ABB RAPID module: PPFP_hurdleJumps

MODULE Weld_ALL_OF_THE_Channels_PR3


    ! NOTES
    ! 6/18/18  CHANGED THE LRnRL_CHAN SETTER's FORLOOP TO START @ 1, WAS MISSING ON M-55's
    ! 3/25/19 CHANGED LL/RR GENERIC STITCH TO SKIP WELD 1 IF ITS A TIGHT BOX
    !  ALSO MADE CHANGES TO THE LRnRL_CHANPLAN, THE_OBJECT = "Push_Stop",   3RD IF TO MAKE THE WELD FLIP IF THE WELD START WAS IN THE MIDDLE OF THE PUSHSTOP
    ! R23  ADDED SR_X2_Y3.TRANS.Y TO THE HURDLES.  TO ALLOW SOME WIGGLE ROOM WHILE TACKING UP, AND STILL BE ABLE TO HOP THE FENCES.
    ! R27 Changed " LRnRL_CHAN_PLAN "Y4"; " FROM "IF (THE_OBJECT = "Y3" AND HORIZ_Y3 <> FP_Height) OR ( THE_OBJECT = "Y4" AND HORIZ_Y4 <> FP_Height) THEN"  TO "IF (THE_OBJECT = "Y3" AND HORIZ_Y3 <> FP_Height) OR ( THE_OBJECT = "Y4" AND HORIZ_Y4 = FP_Height) THEN"
	! 10/21/19 SS
    !  ADDED  " and MY3_Weld_Count > 0 THEN " TO KEEP THE WELD FROM BEING FLIPPED OVER WHEN THERE IS NO CENTER BAR 6/3/20 SS

	! CHANGED PLAN_dUH_cHAN, WHEN W=7, FOR PUSH_STOP = 303,ON 6894640 WAS CRASHING 10/20/20/SS

	! Changed the arrays from 35 to 40, ran out of welds, gave error.  7/22/21/SS

    ! UpDated 7/22/21/SS skipping all weld below the anchor on LRnRL, just to satisify the need of having a AngleIron inside the FP 6898779 on a Friday when I'm not here and Dan W. will just walk away.

PERS robtarget RL_Chan_goingUP:=[[248.58,439.22,15.69],[0.0743186,0.868569,0.302507,0.385428],[0,1,-2,0],[9E+09,-45,0.00451687,9E+09,9E+09,9E+09]];
PERS robtarget RL_Chan_goingUPcorner:=[[248.57,468.99,15.69],[0.00441198,0.818231,0.408605,0.404377],[0,1,-2,0],[9E+09,-40,-5,9E+09,9E+09,9E+09]];

PERS robtarget RL_Chan_goingDOWN:=[[248.55,439.20,15.69],[0.166009,0.884241,0.263964,0.347682],[0,1,-2,0],[9E+09,-45,0.00435694,9E+09,9E+09,9E+09]];
PERS robtarget RL_Chan_BOTTOMcorner:=[[248.55,408.61,15.69],[0.263807,0.884566,0.230134,0.308201],[0,1,-2,0],[9E+09,-40,5.00001,9E+09,9E+09,9E+09]];

PERS robtarget RL_CHANFLAT_goingup:=[[223.12,483.90,15.69],[0.0686406,0.860922,0.436323,0.252434],[0,1,-2,0],[9E+09,-30,0.00345066,9E+09,9E+09,9E+09]];
PERS robtarget RL_CHANFLAT_TOPcorner:=[[223.12,483.90,15.69],[0.0592125,-0.838583,-0.451769,-0.298627],[0,1,-2,0],[9E+09,-25,-4.99996,9E+09,9E+09,9E+09]];

PERS robtarget LL_CHAN_GoingUp:=[[-270.37,436.99,15.21],[0.144124,0.788012,0.487648,0.347081],[0,0,-2,0],[9E+09,-45,0.00410816,9E+09,9E+09,9E+09]];
PERS robtarget LL_CHAN_goingupcorner:=[[-265.50,887.94,15.22],[0.0140209,0.753344,0.518535,0.404224],[-1,0,-1,0],[9E+09,-40,-5,9E+09,9E+09,9E+09]];

PERS robtarget LL_CHAN_GOINGdown:=[[-270.37,436.99,15.21],[0.22246,0.805806,0.454482,0.307627],[0,0,-2,0],[9E+09,-45,0.00410816,9E+09,9E+09,9E+09]];
PERS robtarget LL_CHAN_GOINGdowncorner:=[[-270.36,411.33,15.20],[0.297563,0.81565,0.425985,0.254378],[0,0,-2,0],[9E+09,-40,4.99995,9E+09,9E+09,9E+09]];


PERS robtarget RR_CHAN_GOINGup:=[[265.74,425.05,15.18],[0.346334,0.329821,-0.862433,-0.165773],[-1,0,-2,0],[9E+09,-45,180,9E+09,9E+09,9E+09]];
PERS robtarget RR_CHAN_TOPcorner:=[[265.70,886.67,15.16],[0.257593,0.29389,-0.878079,-0.276138],[-1,0,-2,0],[9E+09,-40,185,9E+09,9E+09,9E+09]];

PERS robtarget RR_CHAN_GOINGdown:=[[269.75,437.02,16.58],[0.403142,0.332329,-0.846748,-0.100255],[-1,0,-2,0],[9E+09,-45,180,9E+09,9E+09,9E+09]];
PERS robtarget RR_CHAN_BOTTOMcorner:=[[269.76,437.02,16.58],[0.430288,0.36564,-0.825086,0.0198048],[-1,0,-1,0],[9E+09,-40,175,9E+09,9E+09,9E+09]];

PERS robtarget LR_CHAN_GOINGup:=[[-249.44,441.38,17.56],[0.34969,0.292965,-0.875927,-0.156972],[-1,0,-2,0],[9E+09,-45,180,9E+09,9E+09,9E+09]];
PERS robtarget LR_CHAN_goingup_corner:=[[-249.44,441.36,17.56],[0.332557,0.268512,-0.875476,-0.225495],[-1,0,-2,0],[9E+09,-40,185,9E+09,9E+09,9E+09]];

PERS robtarget LR_CHAN_GOINGdown:=[[-249.43,441.36,17.56],[0.393213,0.316458,-0.858163,-0.0937788],[-1,0,-2,0],[9E+09,-45,180,9E+09,9E+09,9E+09]];
PERS robtarget LR_CHAN_goingdown_corner:=[[-249.43,441.35,17.56],[0.431123,0.340521,-0.835569,0.0017755],[-1,0,-2,0],[9E+09,-40,175,9E+09,9E+09,9E+09]];

PERS robtarget LR_CHANFLAT_GOINGup:=[[-225.09,482.69,17.56],[0.267219,0.316082,-0.899666,-0.138875],[-1,0,-2,0],[9E+09,-30,180,9E+09,9E+09,9E+09]];
PERS robtarget LR_CHANFLAT_GOINGupcorner:=[[-225.09,482.69,17.56],[0.224093,0.303126,-0.899516,-0.220836],[-1,0,-2,0],[9E+09,-25,185,9E+09,9E+09,9E+09]];




VAR robtarget LL_CHAN_WELDS{40,3}:=[[ [[184.43,695.20,80.98],[0.0842675,0.873996,0.3985,0.265006],[0,0,0,0],[9E+09,-30,0.00423255,9E+09,9E+09,9E+09]],[[184.43,695.20,80.98],[0.0842675,0.873996,0.3985,0.265006],[0,0,0,0],[9E+09,-30,0.00423255,9E+09,9E+09,9E+09]],[[184.43,695.20,80.98],[0.0842675,0.873996,0.3985,0.265006],[0,0,0,0],[9E+09,-30,0.00423255,9E+09,9E+09,9E+09]]],
     [[[184.43,695.20,80.98],[0.0842675,0.873996,0.3985,0.265006],[0,0,0,0],[9E+09,-30,0.00423255,9E+09,9E+09,9E+09]],[[184.43,695.20,80.98],[0.0842675,0.873996,0.3985,0.265006],[0,0,0,0],[9E+09,-30,0.00423255,9E+09,9E+09,9E+09]],[[184.43,695.20,80.98],[0.0842675,0.873996,0.3985,0.265006],[0,0,0,0],[9E+09,-30,0.00423255,9E+09,9E+09,9E+09]]],
     [[[184.43,695.20,80.98],[0.0842675,0.873996,0.3985,0.265006],[0,0,0,0],[9E+09,-30,0.00423255,9E+09,9E+09,9E+09]],[[184.43,695.20,80.98],[0.0842675,0.873996,0.3985,0.265006],[0,0,0,0],[9E+09,-30,0.00423255,9E+09,9E+09,9E+09]],[[184.43,695.20,80.98],[0.0842675,0.873996,0.3985,0.265006],[0,0,0,0],[9E+09,-30,0.00423255,9E+09,9E+09,9E+09]]],
     [[[184.43,695.20,80.98],[0.0842675,0.873996,0.3985,0.265006],[0,0,0,0],[9E+09,-30,0.00423255,9E+09,9E+09,9E+09]],[[184.43,695.20,80.98],[0.0842675,0.873996,0.3985,0.265006],[0,0,0,0],[9E+09,-30,0.00423255,9E+09,9E+09,9E+09]],[[184.43,695.20,80.98],[0.0842675,0.873996,0.3985,0.265006],[0,0,0,0],[9E+09,-30,0.00423255,9E+09,9E+09,9E+09]]],
     [[[184.43,695.20,80.98],[0.0842675,0.873996,0.3985,0.265006],[0,0,0,0],[9E+09,-30,0.00423255,9E+09,9E+09,9E+09]],[[184.43,695.20,80.98],[0.0842675,0.873996,0.3985,0.265006],[0,0,0,0],[9E+09,-30,0.00423255,9E+09,9E+09,9E+09]],[[184.43,695.20,80.98],[0.0842675,0.873996,0.3985,0.265006],[0,0,0,0],[9E+09,-30,0.00423255,9E+09,9E+09,9E+09]]],
     [[[184.43,695.20,80.98],[0.0842675,0.873996,0.3985,0.265006],[0,0,0,0],[9E+09,-30,0.00423255,9E+09,9E+09,9E+09]],[[184.43,695.20,80.98],[0.0842675,0.873996,0.3985,0.265006],[0,0,0,0],[9E+09,-30,0.00423255,9E+09,9E+09,9E+09]],[[184.43,695.20,80.98],[0.0842675,0.873996,0.3985,0.265006],[0,0,0,0],[9E+09,-30,0.00423255,9E+09,9E+09,9E+09]]],
     [[[184.43,695.20,80.98],[0.0842675,0.873996,0.3985,0.265006],[0,0,0,0],[9E+09,-30,0.00423255,9E+09,9E+09,9E+09]],[[184.43,695.20,80.98],[0.0842675,0.873996,0.3985,0.265006],[0,0,0,0],[9E+09,-30,0.00423255,9E+09,9E+09,9E+09]],[[184.43,695.20,80.98],[0.0842675,0.873996,0.3985,0.265006],[0,0,0,0],[9E+09,-30,0.00423255,9E+09,9E+09,9E+09]]],
     [[[184.43,695.20,80.98],[0.0842675,0.873996,0.3985,0.265006],[0,0,0,0],[9E+09,-30,0.00423255,9E+09,9E+09,9E+09]],[[184.43,695.20,80.98],[0.0842675,0.873996,0.3985,0.265006],[0,0,0,0],[9E+09,-30,0.00423255,9E+09,9E+09,9E+09]],[[184.43,695.20,80.98],[0.0842675,0.873996,0.3985,0.265006],[0,0,0,0],[9E+09,-30,0.00423255,9E+09,9E+09,9E+09]]],
     [[[184.43,695.20,80.98],[0.0842675,0.873996,0.3985,0.265006],[0,0,0,0],[9E+09,-30,0.00423255,9E+09,9E+09,9E+09]],[[184.43,695.20,80.98],[0.0842675,0.873996,0.3985,0.265006],[0,0,0,0],[9E+09,-30,0.00423255,9E+09,9E+09,9E+09]],[[184.43,695.20,80.98],[0.0842675,0.873996,0.3985,0.265006],[0,0,0,0],[9E+09,-30,0.00423255,9E+09,9E+09,9E+09]]],
     [[[184.43,695.20,80.98],[0.0842675,0.873996,0.3985,0.265006],[0,0,0,0],[9E+09,-30,0.00423255,9E+09,9E+09,9E+09]],[[184.43,695.20,80.98],[0.0842675,0.873996,0.3985,0.265006],[0,0,0,0],[9E+09,-30,0.00423255,9E+09,9E+09,9E+09]],[[184.43,695.20,80.98],[0.0842675,0.873996,0.3985,0.265006],[0,0,0,0],[9E+09,-30,0.00423255,9E+09,9E+09,9E+09]]],
     [[[184.43,695.20,80.98],[0.0842675,0.873996,0.3985,0.265006],[0,0,0,0],[9E+09,-30,0.00423255,9E+09,9E+09,9E+09]],[[184.43,695.20,80.98],[0.0842675,0.873996,0.3985,0.265006],[0,0,0,0],[9E+09,-30,0.00423255,9E+09,9E+09,9E+09]],[[184.43,695.20,80.98],[0.0842675,0.873996,0.3985,0.265006],[0,0,0,0],[9E+09,-30,0.00423255,9E+09,9E+09,9E+09]]],
     [[[184.43,695.20,80.98],[0.0842675,0.873996,0.3985,0.265006],[0,0,0,0],[9E+09,-30,0.00423255,9E+09,9E+09,9E+09]],[[184.43,695.20,80.98],[0.0842675,0.873996,0.3985,0.265006],[0,0,0,0],[9E+09,-30,0.00423255,9E+09,9E+09,9E+09]],[[184.43,695.20,80.98],[0.0842675,0.873996,0.3985,0.265006],[0,0,0,0],[9E+09,-30,0.00423255,9E+09,9E+09,9E+09]]],
     [[[184.43,695.20,80.98],[0.0842675,0.873996,0.3985,0.265006],[0,0,0,0],[9E+09,-30,0.00423255,9E+09,9E+09,9E+09]],[[184.43,695.20,80.98],[0.0842675,0.873996,0.3985,0.265006],[0,0,0,0],[9E+09,-30,0.00423255,9E+09,9E+09,9E+09]],[[184.43,695.20,80.98],[0.0842675,0.873996,0.3985,0.265006],[0,0,0,0],[9E+09,-30,0.00423255,9E+09,9E+09,9E+09]]],
     [[[184.43,695.20,80.98],[0.0842675,0.873996,0.3985,0.265006],[0,0,0,0],[9E+09,-30,0.00423255,9E+09,9E+09,9E+09]],[[184.43,695.20,80.98],[0.0842675,0.873996,0.3985,0.265006],[0,0,0,0],[9E+09,-30,0.00423255,9E+09,9E+09,9E+09]],[[184.43,695.20,80.98],[0.0842675,0.873996,0.3985,0.265006],[0,0,0,0],[9E+09,-30,0.00423255,9E+09,9E+09,9E+09]]],
     [[[184.43,695.20,80.98],[0.0842675,0.873996,0.3985,0.265006],[0,0,0,0],[9E+09,-30,0.00423255,9E+09,9E+09,9E+09]],[[184.43,695.20,80.98],[0.0842675,0.873996,0.3985,0.265006],[0,0,0,0],[9E+09,-30,0.00423255,9E+09,9E+09,9E+09]],[[184.43,695.20,80.98],[0.0842675,0.873996,0.3985,0.265006],[0,0,0,0],[9E+09,-30,0.00423255,9E+09,9E+09,9E+09]]],
     [[[184.43,695.20,80.98],[0.0842675,0.873996,0.3985,0.265006],[0,0,0,0],[9E+09,-30,0.00423255,9E+09,9E+09,9E+09]],[[184.43,695.20,80.98],[0.0842675,0.873996,0.3985,0.265006],[0,0,0,0],[9E+09,-30,0.00423255,9E+09,9E+09,9E+09]],[[184.43,695.20,80.98],[0.0842675,0.873996,0.3985,0.265006],[0,0,0,0],[9E+09,-30,0.00423255,9E+09,9E+09,9E+09]]],
     [[[184.43,695.20,80.98],[0.0842675,0.873996,0.3985,0.265006],[0,0,0,0],[9E+09,-30,0.00423255,9E+09,9E+09,9E+09]],[[184.43,695.20,80.98],[0.0842675,0.873996,0.3985,0.265006],[0,0,0,0],[9E+09,-30,0.00423255,9E+09,9E+09,9E+09]],[[184.43,695.20,80.98],[0.0842675,0.873996,0.3985,0.265006],[0,0,0,0],[9E+09,-30,0.00423255,9E+09,9E+09,9E+09]]],
     [[[184.43,695.20,80.98],[0.0842675,0.873996,0.3985,0.265006],[0,0,0,0],[9E+09,-30,0.00423255,9E+09,9E+09,9E+09]],[[184.43,695.20,80.98],[0.0842675,0.873996,0.3985,0.265006],[0,0,0,0],[9E+09,-30,0.00423255,9E+09,9E+09,9E+09]],[[184.43,695.20,80.98],[0.0842675,0.873996,0.3985,0.265006],[0,0,0,0],[9E+09,-30,0.00423255,9E+09,9E+09,9E+09]]],
     [[[184.43,695.20,80.98],[0.0842675,0.873996,0.3985,0.265006],[0,0,0,0],[9E+09,-30,0.00423255,9E+09,9E+09,9E+09]],[[184.43,695.20,80.98],[0.0842675,0.873996,0.3985,0.265006],[0,0,0,0],[9E+09,-30,0.00423255,9E+09,9E+09,9E+09]],[[184.43,695.20,80.98],[0.0842675,0.873996,0.3985,0.265006],[0,0,0,0],[9E+09,-30,0.00423255,9E+09,9E+09,9E+09]]],
     [[[184.43,695.20,80.98],[0.0842675,0.873996,0.3985,0.265006],[0,0,0,0],[9E+09,-30,0.00423255,9E+09,9E+09,9E+09]],[[184.43,695.20,80.98],[0.0842675,0.873996,0.3985,0.265006],[0,0,0,0],[9E+09,-30,0.00423255,9E+09,9E+09,9E+09]],[[184.43,695.20,80.98],[0.0842675,0.873996,0.3985,0.265006],[0,0,0,0],[9E+09,-30,0.00423255,9E+09,9E+09,9E+09]]],
     [[[184.43,695.20,80.98],[0.0842675,0.873996,0.3985,0.265006],[0,0,0,0],[9E+09,-30,0.00423255,9E+09,9E+09,9E+09]],[[184.43,695.20,80.98],[0.0842675,0.873996,0.3985,0.265006],[0,0,0,0],[9E+09,-30,0.00423255,9E+09,9E+09,9E+09]],[[184.43,695.20,80.98],[0.0842675,0.873996,0.3985,0.265006],[0,0,0,0],[9E+09,-30,0.00423255,9E+09,9E+09,9E+09]]],
     [[[184.43,695.20,80.98],[0.0842675,0.873996,0.3985,0.265006],[0,0,0,0],[9E+09,-30,0.00423255,9E+09,9E+09,9E+09]],[[184.43,695.20,80.98],[0.0842675,0.873996,0.3985,0.265006],[0,0,0,0],[9E+09,-30,0.00423255,9E+09,9E+09,9E+09]],[[184.43,695.20,80.98],[0.0842675,0.873996,0.3985,0.265006],[0,0,0,0],[9E+09,-30,0.00423255,9E+09,9E+09,9E+09]]],
     [[[184.43,695.20,80.98],[0.0842675,0.873996,0.3985,0.265006],[0,0,0,0],[9E+09,-30,0.00423255,9E+09,9E+09,9E+09]],[[184.43,695.20,80.98],[0.0842675,0.873996,0.3985,0.265006],[0,0,0,0],[9E+09,-30,0.00423255,9E+09,9E+09,9E+09]],[[184.43,695.20,80.98],[0.0842675,0.873996,0.3985,0.265006],[0,0,0,0],[9E+09,-30,0.00423255,9E+09,9E+09,9E+09]]],
     [[[184.43,695.20,80.98],[0.0842675,0.873996,0.3985,0.265006],[0,0,0,0],[9E+09,-30,0.00423255,9E+09,9E+09,9E+09]],[[184.43,695.20,80.98],[0.0842675,0.873996,0.3985,0.265006],[0,0,0,0],[9E+09,-30,0.00423255,9E+09,9E+09,9E+09]],[[184.43,695.20,80.98],[0.0842675,0.873996,0.3985,0.265006],[0,0,0,0],[9E+09,-30,0.00423255,9E+09,9E+09,9E+09]]],
     [[[184.43,695.20,80.98],[0.0842675,0.873996,0.3985,0.265006],[0,0,0,0],[9E+09,-30,0.00423255,9E+09,9E+09,9E+09]],[[184.43,695.20,80.98],[0.0842675,0.873996,0.3985,0.265006],[0,0,0,0],[9E+09,-30,0.00423255,9E+09,9E+09,9E+09]],[[184.43,695.20,80.98],[0.0842675,0.873996,0.3985,0.265006],[0,0,0,0],[9E+09,-30,0.00423255,9E+09,9E+09,9E+09]]],
     [[[184.43,695.20,80.98],[0.0842675,0.873996,0.3985,0.265006],[0,0,0,0],[9E+09,-30,0.00423255,9E+09,9E+09,9E+09]],[[184.43,695.20,80.98],[0.0842675,0.873996,0.3985,0.265006],[0,0,0,0],[9E+09,-30,0.00423255,9E+09,9E+09,9E+09]],[[184.43,695.20,80.98],[0.0842675,0.873996,0.3985,0.265006],[0,0,0,0],[9E+09,-30,0.00423255,9E+09,9E+09,9E+09]]],
     [[[184.43,695.20,80.98],[0.0842675,0.873996,0.3985,0.265006],[0,0,0,0],[9E+09,-30,0.00423255,9E+09,9E+09,9E+09]],[[184.43,695.20,80.98],[0.0842675,0.873996,0.3985,0.265006],[0,0,0,0],[9E+09,-30,0.00423255,9E+09,9E+09,9E+09]],[[184.43,695.20,80.98],[0.0842675,0.873996,0.3985,0.265006],[0,0,0,0],[9E+09,-30,0.00423255,9E+09,9E+09,9E+09]]],
     [[[184.43,695.20,80.98],[0.0842675,0.873996,0.3985,0.265006],[0,0,0,0],[9E+09,-30,0.00423255,9E+09,9E+09,9E+09]],[[184.43,695.20,80.98],[0.0842675,0.873996,0.3985,0.265006],[0,0,0,0],[9E+09,-30,0.00423255,9E+09,9E+09,9E+09]],[[184.43,695.20,80.98],[0.0842675,0.873996,0.3985,0.265006],[0,0,0,0],[9E+09,-30,0.00423255,9E+09,9E+09,9E+09]]],
     [[[184.43,695.20,80.98],[0.0842675,0.873996,0.3985,0.265006],[0,0,0,0],[9E+09,-30,0.00423255,9E+09,9E+09,9E+09]],[[184.43,695.20,80.98],[0.0842675,0.873996,0.3985,0.265006],[0,0,0,0],[9E+09,-30,0.00423255,9E+09,9E+09,9E+09]],[[184.43,695.20,80.98],[0.0842675,0.873996,0.3985,0.265006],[0,0,0,0],[9E+09,-30,0.00423255,9E+09,9E+09,9E+09]]],
     [[[184.43,695.20,80.98],[0.0842675,0.873996,0.3985,0.265006],[0,0,0,0],[9E+09,-30,0.00423255,9E+09,9E+09,9E+09]],[[184.43,695.20,80.98],[0.0842675,0.873996,0.3985,0.265006],[0,0,0,0],[9E+09,-30,0.00423255,9E+09,9E+09,9E+09]],[[184.43,695.20,80.98],[0.0842675,0.873996,0.3985,0.265006],[0,0,0,0],[9E+09,-30,0.00423255,9E+09,9E+09,9E+09]]],
	 [[[184.43,695.20,80.98],[0.0842675,0.873996,0.3985,0.265006],[0,0,0,0],[9E+09,-30,0.00423255,9E+09,9E+09,9E+09]],[[184.43,695.20,80.98],[0.0842675,0.873996,0.3985,0.265006],[0,0,0,0],[9E+09,-30,0.00423255,9E+09,9E+09,9E+09]],[[184.43,695.20,80.98],[0.0842675,0.873996,0.3985,0.265006],[0,0,0,0],[9E+09,-30,0.00423255,9E+09,9E+09,9E+09]]],
     [[[184.43,695.20,80.98],[0.0842675,0.873996,0.3985,0.265006],[0,0,0,0],[9E+09,-30,0.00423255,9E+09,9E+09,9E+09]],[[184.43,695.20,80.98],[0.0842675,0.873996,0.3985,0.265006],[0,0,0,0],[9E+09,-30,0.00423255,9E+09,9E+09,9E+09]],[[184.43,695.20,80.98],[0.0842675,0.873996,0.3985,0.265006],[0,0,0,0],[9E+09,-30,0.00423255,9E+09,9E+09,9E+09]]],
     [[[184.43,695.20,80.98],[0.0842675,0.873996,0.3985,0.265006],[0,0,0,0],[9E+09,-30,0.00423255,9E+09,9E+09,9E+09]],[[184.43,695.20,80.98],[0.0842675,0.873996,0.3985,0.265006],[0,0,0,0],[9E+09,-30,0.00423255,9E+09,9E+09,9E+09]],[[184.43,695.20,80.98],[0.0842675,0.873996,0.3985,0.265006],[0,0,0,0],[9E+09,-30,0.00423255,9E+09,9E+09,9E+09]]],
     [[[184.43,695.20,80.98],[0.0842675,0.873996,0.3985,0.265006],[0,0,0,0],[9E+09,-30,0.00423255,9E+09,9E+09,9E+09]],[[184.43,695.20,80.98],[0.0842675,0.873996,0.3985,0.265006],[0,0,0,0],[9E+09,-30,0.00423255,9E+09,9E+09,9E+09]],[[184.43,695.20,80.98],[0.0842675,0.873996,0.3985,0.265006],[0,0,0,0],[9E+09,-30,0.00423255,9E+09,9E+09,9E+09]]],
     [[[184.43,695.20,80.98],[0.0842675,0.873996,0.3985,0.265006],[0,0,0,0],[9E+09,-30,0.00423255,9E+09,9E+09,9E+09]],[[184.43,695.20,80.98],[0.0842675,0.873996,0.3985,0.265006],[0,0,0,0],[9E+09,-30,0.00423255,9E+09,9E+09,9E+09]],[[184.43,695.20,80.98],[0.0842675,0.873996,0.3985,0.265006],[0,0,0,0],[9E+09,-30,0.00423255,9E+09,9E+09,9E+09]]],
	 [[[184.43,695.20,80.98],[0.0842675,0.873996,0.3985,0.265006],[0,0,0,0],[9E+09,-30,0.00423255,9E+09,9E+09,9E+09]],[[184.43,695.20,80.98],[0.0842675,0.873996,0.3985,0.265006],[0,0,0,0],[9E+09,-30,0.00423255,9E+09,9E+09,9E+09]],[[184.43,695.20,80.98],[0.0842675,0.873996,0.3985,0.265006],[0,0,0,0],[9E+09,-30,0.00423255,9E+09,9E+09,9E+09]]],
     [[[184.43,695.20,80.98],[0.0842675,0.873996,0.3985,0.265006],[0,0,0,0],[9E+09,-30,0.00423255,9E+09,9E+09,9E+09]],[[184.43,695.20,80.98],[0.0842675,0.873996,0.3985,0.265006],[0,0,0,0],[9E+09,-30,0.00423255,9E+09,9E+09,9E+09]],[[184.43,695.20,80.98],[0.0842675,0.873996,0.3985,0.265006],[0,0,0,0],[9E+09,-30,0.00423255,9E+09,9E+09,9E+09]]],
     [[[184.43,695.20,80.98],[0.0842675,0.873996,0.3985,0.265006],[0,0,0,0],[9E+09,-30,0.00423255,9E+09,9E+09,9E+09]],[[184.43,695.20,80.98],[0.0842675,0.873996,0.3985,0.265006],[0,0,0,0],[9E+09,-30,0.00423255,9E+09,9E+09,9E+09]],[[184.43,695.20,80.98],[0.0842675,0.873996,0.3985,0.265006],[0,0,0,0],[9E+09,-30,0.00423255,9E+09,9E+09,9E+09]]],
     [[[184.43,695.20,80.98],[0.0842675,0.873996,0.3985,0.265006],[0,0,0,0],[9E+09,-30,0.00423255,9E+09,9E+09,9E+09]],[[184.43,695.20,80.98],[0.0842675,0.873996,0.3985,0.265006],[0,0,0,0],[9E+09,-30,0.00423255,9E+09,9E+09,9E+09]],[[184.43,695.20,80.98],[0.0842675,0.873996,0.3985,0.265006],[0,0,0,0],[9E+09,-30,0.00423255,9E+09,9E+09,9E+09]]],
     [[[184.43,695.20,80.98],[0.0842675,0.873996,0.3985,0.265006],[0,0,0,0],[9E+09,-30,0.00423255,9E+09,9E+09,9E+09]],[[184.43,695.20,80.98],[0.0842675,0.873996,0.3985,0.265006],[0,0,0,0],[9E+09,-30,0.00423255,9E+09,9E+09,9E+09]],[[184.43,695.20,80.98],[0.0842675,0.873996,0.3985,0.265006],[0,0,0,0],[9E+09,-30,0.00423255,9E+09,9E+09,9E+09]]]];

VAR robtarget LR_CHAN_WELDS{40,3}:=[[ [[184.43,695.20,80.98],[0.0842675,0.873996,0.3985,0.265006],[0,0,0,0],[9E+09,-30,0.00423255,9E+09,9E+09,9E+09]],[[184.43,695.20,80.98],[0.0842675,0.873996,0.3985,0.265006],[0,0,0,0],[9E+09,-30,0.00423255,9E+09,9E+09,9E+09]],[[184.43,695.20,80.98],[0.0842675,0.873996,0.3985,0.265006],[0,0,0,0],[9E+09,-30,0.00423255,9E+09,9E+09,9E+09]]],
     [[[184.43,695.20,80.98],[0.0842675,0.873996,0.3985,0.265006],[0,0,0,0],[9E+09,-30,0.00423255,9E+09,9E+09,9E+09]],[[184.43,695.20,80.98],[0.0842675,0.873996,0.3985,0.265006],[0,0,0,0],[9E+09,-30,0.00423255,9E+09,9E+09,9E+09]],[[184.43,695.20,80.98],[0.0842675,0.873996,0.3985,0.265006],[0,0,0,0],[9E+09,-30,0.00423255,9E+09,9E+09,9E+09]]],
     [[[184.43,695.20,80.98],[0.0842675,0.873996,0.3985,0.265006],[0,0,0,0],[9E+09,-30,0.00423255,9E+09,9E+09,9E+09]],[[184.43,695.20,80.98],[0.0842675,0.873996,0.3985,0.265006],[0,0,0,0],[9E+09,-30,0.00423255,9E+09,9E+09,9E+09]],[[184.43,695.20,80.98],[0.0842675,0.873996,0.3985,0.265006],[0,0,0,0],[9E+09,-30,0.00423255,9E+09,9E+09,9E+09]]],
     [[[184.43,695.20,80.98],[0.0842675,0.873996,0.3985,0.265006],[0,0,0,0],[9E+09,-30,0.00423255,9E+09,9E+09,9E+09]],[[184.43,695.20,80.98],[0.0842675,0.873996,0.3985,0.265006],[0,0,0,0],[9E+09,-30,0.00423255,9E+09,9E+09,9E+09]],[[184.43,695.20,80.98],[0.0842675,0.873996,0.3985,0.265006],[0,0,0,0],[9E+09,-30,0.00423255,9E+09,9E+09,9E+09]]],
     [[[184.43,695.20,80.98],[0.0842675,0.873996,0.3985,0.265006],[0,0,0,0],[9E+09,-30,0.00423255,9E+09,9E+09,9E+09]],[[184.43,695.20,80.98],[0.0842675,0.873996,0.3985,0.265006],[0,0,0,0],[9E+09,-30,0.00423255,9E+09,9E+09,9E+09]],[[184.43,695.20,80.98],[0.0842675,0.873996,0.3985,0.265006],[0,0,0,0],[9E+09,-30,0.00423255,9E+09,9E+09,9E+09]]],
     [[[184.43,695.20,80.98],[0.0842675,0.873996,0.3985,0.265006],[0,0,0,0],[9E+09,-30,0.00423255,9E+09,9E+09,9E+09]],[[184.43,695.20,80.98],[0.0842675,0.873996,0.3985,0.265006],[0,0,0,0],[9E+09,-30,0.00423255,9E+09,9E+09,9E+09]],[[184.43,695.20,80.98],[0.0842675,0.873996,0.3985,0.265006],[0,0,0,0],[9E+09,-30,0.00423255,9E+09,9E+09,9E+09]]],
     [[[184.43,695.20,80.98],[0.0842675,0.873996,0.3985,0.265006],[0,0,0,0],[9E+09,-30,0.00423255,9E+09,9E+09,9E+09]],[[184.43,695.20,80.98],[0.0842675,0.873996,0.3985,0.265006],[0,0,0,0],[9E+09,-30,0.00423255,9E+09,9E+09,9E+09]],[[184.43,695.20,80.98],[0.0842675,0.873996,0.3985,0.265006],[0,0,0,0],[9E+09,-30,0.00423255,9E+09,9E+09,9E+09]]],
     [[[184.43,695.20,80.98],[0.0842675,0.873996,0.3985,0.265006],[0,0,0,0],[9E+09,-30,0.00423255,9E+09,9E+09,9E+09]],[[184.43,695.20,80.98],[0.0842675,0.873996,0.3985,0.265006],[0,0,0,0],[9E+09,-30,0.00423255,9E+09,9E+09,9E+09]],[[184.43,695.20,80.98],[0.0842675,0.873996,0.3985,0.265006],[0,0,0,0],[9E+09,-30,0.00423255,9E+09,9E+09,9E+09]]],
     [[[184.43,695.20,80.98],[0.0842675,0.873996,0.3985,0.265006],[0,0,0,0],[9E+09,-30,0.00423255,9E+09,9E+09,9E+09]],[[184.43,695.20,80.98],[0.0842675,0.873996,0.3985,0.265006],[0,0,0,0],[9E+09,-30,0.00423255,9E+09,9E+09,9E+09]],[[184.43,695.20,80.98],[0.0842675,0.873996,0.3985,0.265006],[0,0,0,0],[9E+09,-30,0.00423255,9E+09,9E+09,9E+09]]],
     [[[184.43,695.20,80.98],[0.0842675,0.873996,0.3985,0.265006],[0,0,0,0],[9E+09,-30,0.00423255,9E+09,9E+09,9E+09]],[[184.43,695.20,80.98],[0.0842675,0.873996,0.3985,0.265006],[0,0,0,0],[9E+09,-30,0.00423255,9E+09,9E+09,9E+09]],[[184.43,695.20,80.98],[0.0842675,0.873996,0.3985,0.265006],[0,0,0,0],[9E+09,-30,0.00423255,9E+09,9E+09,9E+09]]],
     [[[184.43,695.20,80.98],[0.0842675,0.873996,0.3985,0.265006],[0,0,0,0],[9E+09,-30,0.00423255,9E+09,9E+09,9E+09]],[[184.43,695.20,80.98],[0.0842675,0.873996,0.3985,0.265006],[0,0,0,0],[9E+09,-30,0.00423255,9E+09,9E+09,9E+09]],[[184.43,695.20,80.98],[0.0842675,0.873996,0.3985,0.265006],[0,0,0,0],[9E+09,-30,0.00423255,9E+09,9E+09,9E+09]]],
     [[[184.43,695.20,80.98],[0.0842675,0.873996,0.3985,0.265006],[0,0,0,0],[9E+09,-30,0.00423255,9E+09,9E+09,9E+09]],[[184.43,695.20,80.98],[0.0842675,0.873996,0.3985,0.265006],[0,0,0,0],[9E+09,-30,0.00423255,9E+09,9E+09,9E+09]],[[184.43,695.20,80.98],[0.0842675,0.873996,0.3985,0.265006],[0,0,0,0],[9E+09,-30,0.00423255,9E+09,9E+09,9E+09]]],
     [[[184.43,695.20,80.98],[0.0842675,0.873996,0.3985,0.265006],[0,0,0,0],[9E+09,-30,0.00423255,9E+09,9E+09,9E+09]],[[184.43,695.20,80.98],[0.0842675,0.873996,0.3985,0.265006],[0,0,0,0],[9E+09,-30,0.00423255,9E+09,9E+09,9E+09]],[[184.43,695.20,80.98],[0.0842675,0.873996,0.3985,0.265006],[0,0,0,0],[9E+09,-30,0.00423255,9E+09,9E+09,9E+09]]],
     [[[184.43,695.20,80.98],[0.0842675,0.873996,0.3985,0.265006],[0,0,0,0],[9E+09,-30,0.00423255,9E+09,9E+09,9E+09]],[[184.43,695.20,80.98],[0.0842675,0.873996,0.3985,0.265006],[0,0,0,0],[9E+09,-30,0.00423255,9E+09,9E+09,9E+09]],[[184.43,695.20,80.98],[0.0842675,0.873996,0.3985,0.265006],[0,0,0,0],[9E+09,-30,0.00423255,9E+09,9E+09,9E+09]]],
     [[[184.43,695.20,80.98],[0.0842675,0.873996,0.3985,0.265006],[0,0,0,0],[9E+09,-30,0.00423255,9E+09,9E+09,9E+09]],[[184.43,695.20,80.98],[0.0842675,0.873996,0.3985,0.265006],[0,0,0,0],[9E+09,-30,0.00423255,9E+09,9E+09,9E+09]],[[184.43,695.20,80.98],[0.0842675,0.873996,0.3985,0.265006],[0,0,0,0],[9E+09,-30,0.00423255,9E+09,9E+09,9E+09]]],
     [[[184.43,695.20,80.98],[0.0842675,0.873996,0.3985,0.265006],[0,0,0,0],[9E+09,-30,0.00423255,9E+09,9E+09,9E+09]],[[184.43,695.20,80.98],[0.0842675,0.873996,0.3985,0.265006],[0,0,0,0],[9E+09,-30,0.00423255,9E+09,9E+09,9E+09]],[[184.43,695.20,80.98],[0.0842675,0.873996,0.3985,0.265006],[0,0,0,0],[9E+09,-30,0.00423255,9E+09,9E+09,9E+09]]],
     [[[184.43,695.20,80.98],[0.0842675,0.873996,0.3985,0.265006],[0,0,0,0],[9E+09,-30,0.00423255,9E+09,9E+09,9E+09]],[[184.43,695.20,80.98],[0.0842675,0.873996,0.3985,0.265006],[0,0,0,0],[9E+09,-30,0.00423255,9E+09,9E+09,9E+09]],[[184.43,695.20,80.98],[0.0842675,0.873996,0.3985,0.265006],[0,0,0,0],[9E+09,-30,0.00423255,9E+09,9E+09,9E+09]]],
     [[[184.43,695.20,80.98],[0.0842675,0.873996,0.3985,0.265006],[0,0,0,0],[9E+09,-30,0.00423255,9E+09,9E+09,9E+09]],[[184.43,695.20,80.98],[0.0842675,0.873996,0.3985,0.265006],[0,0,0,0],[9E+09,-30,0.00423255,9E+09,9E+09,9E+09]],[[184.43,695.20,80.98],[0.0842675,0.873996,0.3985,0.265006],[0,0,0,0],[9E+09,-30,0.00423255,9E+09,9E+09,9E+09]]],
     [[[184.43,695.20,80.98],[0.0842675,0.873996,0.3985,0.265006],[0,0,0,0],[9E+09,-30,0.00423255,9E+09,9E+09,9E+09]],[[184.43,695.20,80.98],[0.0842675,0.873996,0.3985,0.265006],[0,0,0,0],[9E+09,-30,0.00423255,9E+09,9E+09,9E+09]],[[184.43,695.20,80.98],[0.0842675,0.873996,0.3985,0.265006],[0,0,0,0],[9E+09,-30,0.00423255,9E+09,9E+09,9E+09]]],
     [[[184.43,695.20,80.98],[0.0842675,0.873996,0.3985,0.265006],[0,0,0,0],[9E+09,-30,0.00423255,9E+09,9E+09,9E+09]],[[184.43,695.20,80.98],[0.0842675,0.873996,0.3985,0.265006],[0,0,0,0],[9E+09,-30,0.00423255,9E+09,9E+09,9E+09]],[[184.43,695.20,80.98],[0.0842675,0.873996,0.3985,0.265006],[0,0,0,0],[9E+09,-30,0.00423255,9E+09,9E+09,9E+09]]],
     [[[184.43,695.20,80.98],[0.0842675,0.873996,0.3985,0.265006],[0,0,0,0],[9E+09,-30,0.00423255,9E+09,9E+09,9E+09]],[[184.43,695.20,80.98],[0.0842675,0.873996,0.3985,0.265006],[0,0,0,0],[9E+09,-30,0.00423255,9E+09,9E+09,9E+09]],[[184.43,695.20,80.98],[0.0842675,0.873996,0.3985,0.265006],[0,0,0,0],[9E+09,-30,0.00423255,9E+09,9E+09,9E+09]]],
     [[[184.43,695.20,80.98],[0.0842675,0.873996,0.3985,0.265006],[0,0,0,0],[9E+09,-30,0.00423255,9E+09,9E+09,9E+09]],[[184.43,695.20,80.98],[0.0842675,0.873996,0.3985,0.265006],[0,0,0,0],[9E+09,-30,0.00423255,9E+09,9E+09,9E+09]],[[184.43,695.20,80.98],[0.0842675,0.873996,0.3985,0.265006],[0,0,0,0],[9E+09,-30,0.00423255,9E+09,9E+09,9E+09]]],
     [[[184.43,695.20,80.98],[0.0842675,0.873996,0.3985,0.265006],[0,0,0,0],[9E+09,-30,0.00423255,9E+09,9E+09,9E+09]],[[184.43,695.20,80.98],[0.0842675,0.873996,0.3985,0.265006],[0,0,0,0],[9E+09,-30,0.00423255,9E+09,9E+09,9E+09]],[[184.43,695.20,80.98],[0.0842675,0.873996,0.3985,0.265006],[0,0,0,0],[9E+09,-30,0.00423255,9E+09,9E+09,9E+09]]],
     [[[184.43,695.20,80.98],[0.0842675,0.873996,0.3985,0.265006],[0,0,0,0],[9E+09,-30,0.00423255,9E+09,9E+09,9E+09]],[[184.43,695.20,80.98],[0.0842675,0.873996,0.3985,0.265006],[0,0,0,0],[9E+09,-30,0.00423255,9E+09,9E+09,9E+09]],[[184.43,695.20,80.98],[0.0842675,0.873996,0.3985,0.265006],[0,0,0,0],[9E+09,-30,0.00423255,9E+09,9E+09,9E+09]]],
     [[[184.43,695.20,80.98],[0.0842675,0.873996,0.3985,0.265006],[0,0,0,0],[9E+09,-30,0.00423255,9E+09,9E+09,9E+09]],[[184.43,695.20,80.98],[0.0842675,0.873996,0.3985,0.265006],[0,0,0,0],[9E+09,-30,0.00423255,9E+09,9E+09,9E+09]],[[184.43,695.20,80.98],[0.0842675,0.873996,0.3985,0.265006],[0,0,0,0],[9E+09,-30,0.00423255,9E+09,9E+09,9E+09]]],
     [[[184.43,695.20,80.98],[0.0842675,0.873996,0.3985,0.265006],[0,0,0,0],[9E+09,-30,0.00423255,9E+09,9E+09,9E+09]],[[184.43,695.20,80.98],[0.0842675,0.873996,0.3985,0.265006],[0,0,0,0],[9E+09,-30,0.00423255,9E+09,9E+09,9E+09]],[[184.43,695.20,80.98],[0.0842675,0.873996,0.3985,0.265006],[0,0,0,0],[9E+09,-30,0.00423255,9E+09,9E+09,9E+09]]],
     [[[184.43,695.20,80.98],[0.0842675,0.873996,0.3985,0.265006],[0,0,0,0],[9E+09,-30,0.00423255,9E+09,9E+09,9E+09]],[[184.43,695.20,80.98],[0.0842675,0.873996,0.3985,0.265006],[0,0,0,0],[9E+09,-30,0.00423255,9E+09,9E+09,9E+09]],[[184.43,695.20,80.98],[0.0842675,0.873996,0.3985,0.265006],[0,0,0,0],[9E+09,-30,0.00423255,9E+09,9E+09,9E+09]]],
     [[[184.43,695.20,80.98],[0.0842675,0.873996,0.3985,0.265006],[0,0,0,0],[9E+09,-30,0.00423255,9E+09,9E+09,9E+09]],[[184.43,695.20,80.98],[0.0842675,0.873996,0.3985,0.265006],[0,0,0,0],[9E+09,-30,0.00423255,9E+09,9E+09,9E+09]],[[184.43,695.20,80.98],[0.0842675,0.873996,0.3985,0.265006],[0,0,0,0],[9E+09,-30,0.00423255,9E+09,9E+09,9E+09]]],
     [[[184.43,695.20,80.98],[0.0842675,0.873996,0.3985,0.265006],[0,0,0,0],[9E+09,-30,0.00423255,9E+09,9E+09,9E+09]],[[184.43,695.20,80.98],[0.0842675,0.873996,0.3985,0.265006],[0,0,0,0],[9E+09,-30,0.00423255,9E+09,9E+09,9E+09]],[[184.43,695.20,80.98],[0.0842675,0.873996,0.3985,0.265006],[0,0,0,0],[9E+09,-30,0.00423255,9E+09,9E+09,9E+09]]],
     [[[184.43,695.20,80.98],[0.0842675,0.873996,0.3985,0.265006],[0,0,0,0],[9E+09,-30,0.00423255,9E+09,9E+09,9E+09]],[[184.43,695.20,80.98],[0.0842675,0.873996,0.3985,0.265006],[0,0,0,0],[9E+09,-30,0.00423255,9E+09,9E+09,9E+09]],[[184.43,695.20,80.98],[0.0842675,0.873996,0.3985,0.265006],[0,0,0,0],[9E+09,-30,0.00423255,9E+09,9E+09,9E+09]]],
	 [[[184.43,695.20,80.98],[0.0842675,0.873996,0.3985,0.265006],[0,0,0,0],[9E+09,-30,0.00423255,9E+09,9E+09,9E+09]],[[184.43,695.20,80.98],[0.0842675,0.873996,0.3985,0.265006],[0,0,0,0],[9E+09,-30,0.00423255,9E+09,9E+09,9E+09]],[[184.43,695.20,80.98],[0.0842675,0.873996,0.3985,0.265006],[0,0,0,0],[9E+09,-30,0.00423255,9E+09,9E+09,9E+09]]],
     [[[184.43,695.20,80.98],[0.0842675,0.873996,0.3985,0.265006],[0,0,0,0],[9E+09,-30,0.00423255,9E+09,9E+09,9E+09]],[[184.43,695.20,80.98],[0.0842675,0.873996,0.3985,0.265006],[0,0,0,0],[9E+09,-30,0.00423255,9E+09,9E+09,9E+09]],[[184.43,695.20,80.98],[0.0842675,0.873996,0.3985,0.265006],[0,0,0,0],[9E+09,-30,0.00423255,9E+09,9E+09,9E+09]]],
     [[[184.43,695.20,80.98],[0.0842675,0.873996,0.3985,0.265006],[0,0,0,0],[9E+09,-30,0.00423255,9E+09,9E+09,9E+09]],[[184.43,695.20,80.98],[0.0842675,0.873996,0.3985,0.265006],[0,0,0,0],[9E+09,-30,0.00423255,9E+09,9E+09,9E+09]],[[184.43,695.20,80.98],[0.0842675,0.873996,0.3985,0.265006],[0,0,0,0],[9E+09,-30,0.00423255,9E+09,9E+09,9E+09]]],
     [[[184.43,695.20,80.98],[0.0842675,0.873996,0.3985,0.265006],[0,0,0,0],[9E+09,-30,0.00423255,9E+09,9E+09,9E+09]],[[184.43,695.20,80.98],[0.0842675,0.873996,0.3985,0.265006],[0,0,0,0],[9E+09,-30,0.00423255,9E+09,9E+09,9E+09]],[[184.43,695.20,80.98],[0.0842675,0.873996,0.3985,0.265006],[0,0,0,0],[9E+09,-30,0.00423255,9E+09,9E+09,9E+09]]],
     [[[184.43,695.20,80.98],[0.0842675,0.873996,0.3985,0.265006],[0,0,0,0],[9E+09,-30,0.00423255,9E+09,9E+09,9E+09]],[[184.43,695.20,80.98],[0.0842675,0.873996,0.3985,0.265006],[0,0,0,0],[9E+09,-30,0.00423255,9E+09,9E+09,9E+09]],[[184.43,695.20,80.98],[0.0842675,0.873996,0.3985,0.265006],[0,0,0,0],[9E+09,-30,0.00423255,9E+09,9E+09,9E+09]]],
	 [[[184.43,695.20,80.98],[0.0842675,0.873996,0.3985,0.265006],[0,0,0,0],[9E+09,-30,0.00423255,9E+09,9E+09,9E+09]],[[184.43,695.20,80.98],[0.0842675,0.873996,0.3985,0.265006],[0,0,0,0],[9E+09,-30,0.00423255,9E+09,9E+09,9E+09]],[[184.43,695.20,80.98],[0.0842675,0.873996,0.3985,0.265006],[0,0,0,0],[9E+09,-30,0.00423255,9E+09,9E+09,9E+09]]],
     [[[184.43,695.20,80.98],[0.0842675,0.873996,0.3985,0.265006],[0,0,0,0],[9E+09,-30,0.00423255,9E+09,9E+09,9E+09]],[[184.43,695.20,80.98],[0.0842675,0.873996,0.3985,0.265006],[0,0,0,0],[9E+09,-30,0.00423255,9E+09,9E+09,9E+09]],[[184.43,695.20,80.98],[0.0842675,0.873996,0.3985,0.265006],[0,0,0,0],[9E+09,-30,0.00423255,9E+09,9E+09,9E+09]]],
     [[[184.43,695.20,80.98],[0.0842675,0.873996,0.3985,0.265006],[0,0,0,0],[9E+09,-30,0.00423255,9E+09,9E+09,9E+09]],[[184.43,695.20,80.98],[0.0842675,0.873996,0.3985,0.265006],[0,0,0,0],[9E+09,-30,0.00423255,9E+09,9E+09,9E+09]],[[184.43,695.20,80.98],[0.0842675,0.873996,0.3985,0.265006],[0,0,0,0],[9E+09,-30,0.00423255,9E+09,9E+09,9E+09]]],
     [[[184.43,695.20,80.98],[0.0842675,0.873996,0.3985,0.265006],[0,0,0,0],[9E+09,-30,0.00423255,9E+09,9E+09,9E+09]],[[184.43,695.20,80.98],[0.0842675,0.873996,0.3985,0.265006],[0,0,0,0],[9E+09,-30,0.00423255,9E+09,9E+09,9E+09]],[[184.43,695.20,80.98],[0.0842675,0.873996,0.3985,0.265006],[0,0,0,0],[9E+09,-30,0.00423255,9E+09,9E+09,9E+09]]],
     [[[184.43,695.20,80.98],[0.0842675,0.873996,0.3985,0.265006],[0,0,0,0],[9E+09,-30,0.00423255,9E+09,9E+09,9E+09]],[[184.43,695.20,80.98],[0.0842675,0.873996,0.3985,0.265006],[0,0,0,0],[9E+09,-30,0.00423255,9E+09,9E+09,9E+09]],[[184.43,695.20,80.98],[0.0842675,0.873996,0.3985,0.265006],[0,0,0,0],[9E+09,-30,0.00423255,9E+09,9E+09,9E+09]]]];

VAR robtarget RL_CHAN_WELDS{40,3}:=[[ [[184.43,695.20,80.98],[0.0842675,0.873996,0.3985,0.265006],[0,0,0,0],[9E+09,-30,0.00423255,9E+09,9E+09,9E+09]],[[184.43,695.20,80.98],[0.0842675,0.873996,0.3985,0.265006],[0,0,0,0],[9E+09,-30,0.00423255,9E+09,9E+09,9E+09]],[[184.43,695.20,80.98],[0.0842675,0.873996,0.3985,0.265006],[0,0,0,0],[9E+09,-30,0.00423255,9E+09,9E+09,9E+09]]],
     [[[184.43,695.20,80.98],[0.0842675,0.873996,0.3985,0.265006],[0,0,0,0],[9E+09,-30,0.00423255,9E+09,9E+09,9E+09]],[[184.43,695.20,80.98],[0.0842675,0.873996,0.3985,0.265006],[0,0,0,0],[9E+09,-30,0.00423255,9E+09,9E+09,9E+09]],[[184.43,695.20,80.98],[0.0842675,0.873996,0.3985,0.265006],[0,0,0,0],[9E+09,-30,0.00423255,9E+09,9E+09,9E+09]]],
     [[[184.43,695.20,80.98],[0.0842675,0.873996,0.3985,0.265006],[0,0,0,0],[9E+09,-30,0.00423255,9E+09,9E+09,9E+09]],[[184.43,695.20,80.98],[0.0842675,0.873996,0.3985,0.265006],[0,0,0,0],[9E+09,-30,0.00423255,9E+09,9E+09,9E+09]],[[184.43,695.20,80.98],[0.0842675,0.873996,0.3985,0.265006],[0,0,0,0],[9E+09,-30,0.00423255,9E+09,9E+09,9E+09]]],
     [[[184.43,695.20,80.98],[0.0842675,0.873996,0.3985,0.265006],[0,0,0,0],[9E+09,-30,0.00423255,9E+09,9E+09,9E+09]],[[184.43,695.20,80.98],[0.0842675,0.873996,0.3985,0.265006],[0,0,0,0],[9E+09,-30,0.00423255,9E+09,9E+09,9E+09]],[[184.43,695.20,80.98],[0.0842675,0.873996,0.3985,0.265006],[0,0,0,0],[9E+09,-30,0.00423255,9E+09,9E+09,9E+09]]],
     [[[184.43,695.20,80.98],[0.0842675,0.873996,0.3985,0.265006],[0,0,0,0],[9E+09,-30,0.00423255,9E+09,9E+09,9E+09]],[[184.43,695.20,80.98],[0.0842675,0.873996,0.3985,0.265006],[0,0,0,0],[9E+09,-30,0.00423255,9E+09,9E+09,9E+09]],[[184.43,695.20,80.98],[0.0842675,0.873996,0.3985,0.265006],[0,0,0,0],[9E+09,-30,0.00423255,9E+09,9E+09,9E+09]]],
     [[[184.43,695.20,80.98],[0.0842675,0.873996,0.3985,0.265006],[0,0,0,0],[9E+09,-30,0.00423255,9E+09,9E+09,9E+09]],[[184.43,695.20,80.98],[0.0842675,0.873996,0.3985,0.265006],[0,0,0,0],[9E+09,-30,0.00423255,9E+09,9E+09,9E+09]],[[184.43,695.20,80.98],[0.0842675,0.873996,0.3985,0.265006],[0,0,0,0],[9E+09,-30,0.00423255,9E+09,9E+09,9E+09]]],
     [[[184.43,695.20,80.98],[0.0842675,0.873996,0.3985,0.265006],[0,0,0,0],[9E+09,-30,0.00423255,9E+09,9E+09,9E+09]],[[184.43,695.20,80.98],[0.0842675,0.873996,0.3985,0.265006],[0,0,0,0],[9E+09,-30,0.00423255,9E+09,9E+09,9E+09]],[[184.43,695.20,80.98],[0.0842675,0.873996,0.3985,0.265006],[0,0,0,0],[9E+09,-30,0.00423255,9E+09,9E+09,9E+09]]],
     [[[184.43,695.20,80.98],[0.0842675,0.873996,0.3985,0.265006],[0,0,0,0],[9E+09,-30,0.00423255,9E+09,9E+09,9E+09]],[[184.43,695.20,80.98],[0.0842675,0.873996,0.3985,0.265006],[0,0,0,0],[9E+09,-30,0.00423255,9E+09,9E+09,9E+09]],[[184.43,695.20,80.98],[0.0842675,0.873996,0.3985,0.265006],[0,0,0,0],[9E+09,-30,0.00423255,9E+09,9E+09,9E+09]]],
     [[[184.43,695.20,80.98],[0.0842675,0.873996,0.3985,0.265006],[0,0,0,0],[9E+09,-30,0.00423255,9E+09,9E+09,9E+09]],[[184.43,695.20,80.98],[0.0842675,0.873996,0.3985,0.265006],[0,0,0,0],[9E+09,-30,0.00423255,9E+09,9E+09,9E+09]],[[184.43,695.20,80.98],[0.0842675,0.873996,0.3985,0.265006],[0,0,0,0],[9E+09,-30,0.00423255,9E+09,9E+09,9E+09]]],
     [[[184.43,695.20,80.98],[0.0842675,0.873996,0.3985,0.265006],[0,0,0,0],[9E+09,-30,0.00423255,9E+09,9E+09,9E+09]],[[184.43,695.20,80.98],[0.0842675,0.873996,0.3985,0.265006],[0,0,0,0],[9E+09,-30,0.00423255,9E+09,9E+09,9E+09]],[[184.43,695.20,80.98],[0.0842675,0.873996,0.3985,0.265006],[0,0,0,0],[9E+09,-30,0.00423255,9E+09,9E+09,9E+09]]],
     [[[184.43,695.20,80.98],[0.0842675,0.873996,0.3985,0.265006],[0,0,0,0],[9E+09,-30,0.00423255,9E+09,9E+09,9E+09]],[[184.43,695.20,80.98],[0.0842675,0.873996,0.3985,0.265006],[0,0,0,0],[9E+09,-30,0.00423255,9E+09,9E+09,9E+09]],[[184.43,695.20,80.98],[0.0842675,0.873996,0.3985,0.265006],[0,0,0,0],[9E+09,-30,0.00423255,9E+09,9E+09,9E+09]]],
     [[[184.43,695.20,80.98],[0.0842675,0.873996,0.3985,0.265006],[0,0,0,0],[9E+09,-30,0.00423255,9E+09,9E+09,9E+09]],[[184.43,695.20,80.98],[0.0842675,0.873996,0.3985,0.265006],[0,0,0,0],[9E+09,-30,0.00423255,9E+09,9E+09,9E+09]],[[184.43,695.20,80.98],[0.0842675,0.873996,0.3985,0.265006],[0,0,0,0],[9E+09,-30,0.00423255,9E+09,9E+09,9E+09]]],
     [[[184.43,695.20,80.98],[0.0842675,0.873996,0.3985,0.265006],[0,0,0,0],[9E+09,-30,0.00423255,9E+09,9E+09,9E+09]],[[184.43,695.20,80.98],[0.0842675,0.873996,0.3985,0.265006],[0,0,0,0],[9E+09,-30,0.00423255,9E+09,9E+09,9E+09]],[[184.43,695.20,80.98],[0.0842675,0.873996,0.3985,0.265006],[0,0,0,0],[9E+09,-30,0.00423255,9E+09,9E+09,9E+09]]],
     [[[184.43,695.20,80.98],[0.0842675,0.873996,0.3985,0.265006],[0,0,0,0],[9E+09,-30,0.00423255,9E+09,9E+09,9E+09]],[[184.43,695.20,80.98],[0.0842675,0.873996,0.3985,0.265006],[0,0,0,0],[9E+09,-30,0.00423255,9E+09,9E+09,9E+09]],[[184.43,695.20,80.98],[0.0842675,0.873996,0.3985,0.265006],[0,0,0,0],[9E+09,-30,0.00423255,9E+09,9E+09,9E+09]]],
     [[[184.43,695.20,80.98],[0.0842675,0.873996,0.3985,0.265006],[0,0,0,0],[9E+09,-30,0.00423255,9E+09,9E+09,9E+09]],[[184.43,695.20,80.98],[0.0842675,0.873996,0.3985,0.265006],[0,0,0,0],[9E+09,-30,0.00423255,9E+09,9E+09,9E+09]],[[184.43,695.20,80.98],[0.0842675,0.873996,0.3985,0.265006],[0,0,0,0],[9E+09,-30,0.00423255,9E+09,9E+09,9E+09]]],
     [[[184.43,695.20,80.98],[0.0842675,0.873996,0.3985,0.265006],[0,0,0,0],[9E+09,-30,0.00423255,9E+09,9E+09,9E+09]],[[184.43,695.20,80.98],[0.0842675,0.873996,0.3985,0.265006],[0,0,0,0],[9E+09,-30,0.00423255,9E+09,9E+09,9E+09]],[[184.43,695.20,80.98],[0.0842675,0.873996,0.3985,0.265006],[0,0,0,0],[9E+09,-30,0.00423255,9E+09,9E+09,9E+09]]],
     [[[184.43,695.20,80.98],[0.0842675,0.873996,0.3985,0.265006],[0,0,0,0],[9E+09,-30,0.00423255,9E+09,9E+09,9E+09]],[[184.43,695.20,80.98],[0.0842675,0.873996,0.3985,0.265006],[0,0,0,0],[9E+09,-30,0.00423255,9E+09,9E+09,9E+09]],[[184.43,695.20,80.98],[0.0842675,0.873996,0.3985,0.265006],[0,0,0,0],[9E+09,-30,0.00423255,9E+09,9E+09,9E+09]]],
     [[[184.43,695.20,80.98],[0.0842675,0.873996,0.3985,0.265006],[0,0,0,0],[9E+09,-30,0.00423255,9E+09,9E+09,9E+09]],[[184.43,695.20,80.98],[0.0842675,0.873996,0.3985,0.265006],[0,0,0,0],[9E+09,-30,0.00423255,9E+09,9E+09,9E+09]],[[184.43,695.20,80.98],[0.0842675,0.873996,0.3985,0.265006],[0,0,0,0],[9E+09,-30,0.00423255,9E+09,9E+09,9E+09]]],
     [[[184.43,695.20,80.98],[0.0842675,0.873996,0.3985,0.265006],[0,0,0,0],[9E+09,-30,0.00423255,9E+09,9E+09,9E+09]],[[184.43,695.20,80.98],[0.0842675,0.873996,0.3985,0.265006],[0,0,0,0],[9E+09,-30,0.00423255,9E+09,9E+09,9E+09]],[[184.43,695.20,80.98],[0.0842675,0.873996,0.3985,0.265006],[0,0,0,0],[9E+09,-30,0.00423255,9E+09,9E+09,9E+09]]],
     [[[184.43,695.20,80.98],[0.0842675,0.873996,0.3985,0.265006],[0,0,0,0],[9E+09,-30,0.00423255,9E+09,9E+09,9E+09]],[[184.43,695.20,80.98],[0.0842675,0.873996,0.3985,0.265006],[0,0,0,0],[9E+09,-30,0.00423255,9E+09,9E+09,9E+09]],[[184.43,695.20,80.98],[0.0842675,0.873996,0.3985,0.265006],[0,0,0,0],[9E+09,-30,0.00423255,9E+09,9E+09,9E+09]]],
     [[[184.43,695.20,80.98],[0.0842675,0.873996,0.3985,0.265006],[0,0,0,0],[9E+09,-30,0.00423255,9E+09,9E+09,9E+09]],[[184.43,695.20,80.98],[0.0842675,0.873996,0.3985,0.265006],[0,0,0,0],[9E+09,-30,0.00423255,9E+09,9E+09,9E+09]],[[184.43,695.20,80.98],[0.0842675,0.873996,0.3985,0.265006],[0,0,0,0],[9E+09,-30,0.00423255,9E+09,9E+09,9E+09]]],
     [[[184.43,695.20,80.98],[0.0842675,0.873996,0.3985,0.265006],[0,0,0,0],[9E+09,-30,0.00423255,9E+09,9E+09,9E+09]],[[184.43,695.20,80.98],[0.0842675,0.873996,0.3985,0.265006],[0,0,0,0],[9E+09,-30,0.00423255,9E+09,9E+09,9E+09]],[[184.43,695.20,80.98],[0.0842675,0.873996,0.3985,0.265006],[0,0,0,0],[9E+09,-30,0.00423255,9E+09,9E+09,9E+09]]],
     [[[184.43,695.20,80.98],[0.0842675,0.873996,0.3985,0.265006],[0,0,0,0],[9E+09,-30,0.00423255,9E+09,9E+09,9E+09]],[[184.43,695.20,80.98],[0.0842675,0.873996,0.3985,0.265006],[0,0,0,0],[9E+09,-30,0.00423255,9E+09,9E+09,9E+09]],[[184.43,695.20,80.98],[0.0842675,0.873996,0.3985,0.265006],[0,0,0,0],[9E+09,-30,0.00423255,9E+09,9E+09,9E+09]]],
     [[[184.43,695.20,80.98],[0.0842675,0.873996,0.3985,0.265006],[0,0,0,0],[9E+09,-30,0.00423255,9E+09,9E+09,9E+09]],[[184.43,695.20,80.98],[0.0842675,0.873996,0.3985,0.265006],[0,0,0,0],[9E+09,-30,0.00423255,9E+09,9E+09,9E+09]],[[184.43,695.20,80.98],[0.0842675,0.873996,0.3985,0.265006],[0,0,0,0],[9E+09,-30,0.00423255,9E+09,9E+09,9E+09]]],
     [[[184.43,695.20,80.98],[0.0842675,0.873996,0.3985,0.265006],[0,0,0,0],[9E+09,-30,0.00423255,9E+09,9E+09,9E+09]],[[184.43,695.20,80.98],[0.0842675,0.873996,0.3985,0.265006],[0,0,0,0],[9E+09,-30,0.00423255,9E+09,9E+09,9E+09]],[[184.43,695.20,80.98],[0.0842675,0.873996,0.3985,0.265006],[0,0,0,0],[9E+09,-30,0.00423255,9E+09,9E+09,9E+09]]],
     [[[184.43,695.20,80.98],[0.0842675,0.873996,0.3985,0.265006],[0,0,0,0],[9E+09,-30,0.00423255,9E+09,9E+09,9E+09]],[[184.43,695.20,80.98],[0.0842675,0.873996,0.3985,0.265006],[0,0,0,0],[9E+09,-30,0.00423255,9E+09,9E+09,9E+09]],[[184.43,695.20,80.98],[0.0842675,0.873996,0.3985,0.265006],[0,0,0,0],[9E+09,-30,0.00423255,9E+09,9E+09,9E+09]]],
     [[[184.43,695.20,80.98],[0.0842675,0.873996,0.3985,0.265006],[0,0,0,0],[9E+09,-30,0.00423255,9E+09,9E+09,9E+09]],[[184.43,695.20,80.98],[0.0842675,0.873996,0.3985,0.265006],[0,0,0,0],[9E+09,-30,0.00423255,9E+09,9E+09,9E+09]],[[184.43,695.20,80.98],[0.0842675,0.873996,0.3985,0.265006],[0,0,0,0],[9E+09,-30,0.00423255,9E+09,9E+09,9E+09]]],
     [[[184.43,695.20,80.98],[0.0842675,0.873996,0.3985,0.265006],[0,0,0,0],[9E+09,-30,0.00423255,9E+09,9E+09,9E+09]],[[184.43,695.20,80.98],[0.0842675,0.873996,0.3985,0.265006],[0,0,0,0],[9E+09,-30,0.00423255,9E+09,9E+09,9E+09]],[[184.43,695.20,80.98],[0.0842675,0.873996,0.3985,0.265006],[0,0,0,0],[9E+09,-30,0.00423255,9E+09,9E+09,9E+09]]],
     [[[184.43,695.20,80.98],[0.0842675,0.873996,0.3985,0.265006],[0,0,0,0],[9E+09,-30,0.00423255,9E+09,9E+09,9E+09]],[[184.43,695.20,80.98],[0.0842675,0.873996,0.3985,0.265006],[0,0,0,0],[9E+09,-30,0.00423255,9E+09,9E+09,9E+09]],[[184.43,695.20,80.98],[0.0842675,0.873996,0.3985,0.265006],[0,0,0,0],[9E+09,-30,0.00423255,9E+09,9E+09,9E+09]]],
     [[[184.43,695.20,80.98],[0.0842675,0.873996,0.3985,0.265006],[0,0,0,0],[9E+09,-30,0.00423255,9E+09,9E+09,9E+09]],[[184.43,695.20,80.98],[0.0842675,0.873996,0.3985,0.265006],[0,0,0,0],[9E+09,-30,0.00423255,9E+09,9E+09,9E+09]],[[184.43,695.20,80.98],[0.0842675,0.873996,0.3985,0.265006],[0,0,0,0],[9E+09,-30,0.00423255,9E+09,9E+09,9E+09]]],
	 [[[184.43,695.20,80.98],[0.0842675,0.873996,0.3985,0.265006],[0,0,0,0],[9E+09,-30,0.00423255,9E+09,9E+09,9E+09]],[[184.43,695.20,80.98],[0.0842675,0.873996,0.3985,0.265006],[0,0,0,0],[9E+09,-30,0.00423255,9E+09,9E+09,9E+09]],[[184.43,695.20,80.98],[0.0842675,0.873996,0.3985,0.265006],[0,0,0,0],[9E+09,-30,0.00423255,9E+09,9E+09,9E+09]]],
     [[[184.43,695.20,80.98],[0.0842675,0.873996,0.3985,0.265006],[0,0,0,0],[9E+09,-30,0.00423255,9E+09,9E+09,9E+09]],[[184.43,695.20,80.98],[0.0842675,0.873996,0.3985,0.265006],[0,0,0,0],[9E+09,-30,0.00423255,9E+09,9E+09,9E+09]],[[184.43,695.20,80.98],[0.0842675,0.873996,0.3985,0.265006],[0,0,0,0],[9E+09,-30,0.00423255,9E+09,9E+09,9E+09]]],
     [[[184.43,695.20,80.98],[0.0842675,0.873996,0.3985,0.265006],[0,0,0,0],[9E+09,-30,0.00423255,9E+09,9E+09,9E+09]],[[184.43,695.20,80.98],[0.0842675,0.873996,0.3985,0.265006],[0,0,0,0],[9E+09,-30,0.00423255,9E+09,9E+09,9E+09]],[[184.43,695.20,80.98],[0.0842675,0.873996,0.3985,0.265006],[0,0,0,0],[9E+09,-30,0.00423255,9E+09,9E+09,9E+09]]],
     [[[184.43,695.20,80.98],[0.0842675,0.873996,0.3985,0.265006],[0,0,0,0],[9E+09,-30,0.00423255,9E+09,9E+09,9E+09]],[[184.43,695.20,80.98],[0.0842675,0.873996,0.3985,0.265006],[0,0,0,0],[9E+09,-30,0.00423255,9E+09,9E+09,9E+09]],[[184.43,695.20,80.98],[0.0842675,0.873996,0.3985,0.265006],[0,0,0,0],[9E+09,-30,0.00423255,9E+09,9E+09,9E+09]]],
     [[[184.43,695.20,80.98],[0.0842675,0.873996,0.3985,0.265006],[0,0,0,0],[9E+09,-30,0.00423255,9E+09,9E+09,9E+09]],[[184.43,695.20,80.98],[0.0842675,0.873996,0.3985,0.265006],[0,0,0,0],[9E+09,-30,0.00423255,9E+09,9E+09,9E+09]],[[184.43,695.20,80.98],[0.0842675,0.873996,0.3985,0.265006],[0,0,0,0],[9E+09,-30,0.00423255,9E+09,9E+09,9E+09]]],
     [[[184.43,695.20,80.98],[0.0842675,0.873996,0.3985,0.265006],[0,0,0,0],[9E+09,-30,0.00423255,9E+09,9E+09,9E+09]],[[184.43,695.20,80.98],[0.0842675,0.873996,0.3985,0.265006],[0,0,0,0],[9E+09,-30,0.00423255,9E+09,9E+09,9E+09]],[[184.43,695.20,80.98],[0.0842675,0.873996,0.3985,0.265006],[0,0,0,0],[9E+09,-30,0.00423255,9E+09,9E+09,9E+09]]],
     [[[184.43,695.20,80.98],[0.0842675,0.873996,0.3985,0.265006],[0,0,0,0],[9E+09,-30,0.00423255,9E+09,9E+09,9E+09]],[[184.43,695.20,80.98],[0.0842675,0.873996,0.3985,0.265006],[0,0,0,0],[9E+09,-30,0.00423255,9E+09,9E+09,9E+09]],[[184.43,695.20,80.98],[0.0842675,0.873996,0.3985,0.265006],[0,0,0,0],[9E+09,-30,0.00423255,9E+09,9E+09,9E+09]]],
     [[[184.43,695.20,80.98],[0.0842675,0.873996,0.3985,0.265006],[0,0,0,0],[9E+09,-30,0.00423255,9E+09,9E+09,9E+09]],[[184.43,695.20,80.98],[0.0842675,0.873996,0.3985,0.265006],[0,0,0,0],[9E+09,-30,0.00423255,9E+09,9E+09,9E+09]],[[184.43,695.20,80.98],[0.0842675,0.873996,0.3985,0.265006],[0,0,0,0],[9E+09,-30,0.00423255,9E+09,9E+09,9E+09]]],
     [[[184.43,695.20,80.98],[0.0842675,0.873996,0.3985,0.265006],[0,0,0,0],[9E+09,-30,0.00423255,9E+09,9E+09,9E+09]],[[184.43,695.20,80.98],[0.0842675,0.873996,0.3985,0.265006],[0,0,0,0],[9E+09,-30,0.00423255,9E+09,9E+09,9E+09]],[[184.43,695.20,80.98],[0.0842675,0.873996,0.3985,0.265006],[0,0,0,0],[9E+09,-30,0.00423255,9E+09,9E+09,9E+09]]],
     [[[184.43,695.20,80.98],[0.0842675,0.873996,0.3985,0.265006],[0,0,0,0],[9E+09,-30,0.00423255,9E+09,9E+09,9E+09]],[[184.43,695.20,80.98],[0.0842675,0.873996,0.3985,0.265006],[0,0,0,0],[9E+09,-30,0.00423255,9E+09,9E+09,9E+09]],[[184.43,695.20,80.98],[0.0842675,0.873996,0.3985,0.265006],[0,0,0,0],[9E+09,-30,0.00423255,9E+09,9E+09,9E+09]]]];

VAR robtarget RR_CHAN_WELDS{40,3}:=[[ [[184.43,695.20,80.98],[0.0842675,0.873996,0.3985,0.265006],[0,0,0,0],[9E+09,-30,0.00423255,9E+09,9E+09,9E+09]],[[184.43,695.20,80.98],[0.0842675,0.873996,0.3985,0.265006],[0,0,0,0],[9E+09,-30,0.00423255,9E+09,9E+09,9E+09]],[[184.43,695.20,80.98],[0.0842675,0.873996,0.3985,0.265006],[0,0,0,0],[9E+09,-30,0.00423255,9E+09,9E+09,9E+09]]],
     [[[184.43,695.20,80.98],[0.0842675,0.873996,0.3985,0.265006],[0,0,0,0],[9E+09,-30,0.00423255,9E+09,9E+09,9E+09]],[[184.43,695.20,80.98],[0.0842675,0.873996,0.3985,0.265006],[0,0,0,0],[9E+09,-30,0.00423255,9E+09,9E+09,9E+09]],[[184.43,695.20,80.98],[0.0842675,0.873996,0.3985,0.265006],[0,0,0,0],[9E+09,-30,0.00423255,9E+09,9E+09,9E+09]]],
     [[[184.43,695.20,80.98],[0.0842675,0.873996,0.3985,0.265006],[0,0,0,0],[9E+09,-30,0.00423255,9E+09,9E+09,9E+09]],[[184.43,695.20,80.98],[0.0842675,0.873996,0.3985,0.265006],[0,0,0,0],[9E+09,-30,0.00423255,9E+09,9E+09,9E+09]],[[184.43,695.20,80.98],[0.0842675,0.873996,0.3985,0.265006],[0,0,0,0],[9E+09,-30,0.00423255,9E+09,9E+09,9E+09]]],
     [[[184.43,695.20,80.98],[0.0842675,0.873996,0.3985,0.265006],[0,0,0,0],[9E+09,-30,0.00423255,9E+09,9E+09,9E+09]],[[184.43,695.20,80.98],[0.0842675,0.873996,0.3985,0.265006],[0,0,0,0],[9E+09,-30,0.00423255,9E+09,9E+09,9E+09]],[[184.43,695.20,80.98],[0.0842675,0.873996,0.3985,0.265006],[0,0,0,0],[9E+09,-30,0.00423255,9E+09,9E+09,9E+09]]],
     [[[184.43,695.20,80.98],[0.0842675,0.873996,0.3985,0.265006],[0,0,0,0],[9E+09,-30,0.00423255,9E+09,9E+09,9E+09]],[[184.43,695.20,80.98],[0.0842675,0.873996,0.3985,0.265006],[0,0,0,0],[9E+09,-30,0.00423255,9E+09,9E+09,9E+09]],[[184.43,695.20,80.98],[0.0842675,0.873996,0.3985,0.265006],[0,0,0,0],[9E+09,-30,0.00423255,9E+09,9E+09,9E+09]]],
     [[[184.43,695.20,80.98],[0.0842675,0.873996,0.3985,0.265006],[0,0,0,0],[9E+09,-30,0.00423255,9E+09,9E+09,9E+09]],[[184.43,695.20,80.98],[0.0842675,0.873996,0.3985,0.265006],[0,0,0,0],[9E+09,-30,0.00423255,9E+09,9E+09,9E+09]],[[184.43,695.20,80.98],[0.0842675,0.873996,0.3985,0.265006],[0,0,0,0],[9E+09,-30,0.00423255,9E+09,9E+09,9E+09]]],
     [[[184.43,695.20,80.98],[0.0842675,0.873996,0.3985,0.265006],[0,0,0,0],[9E+09,-30,0.00423255,9E+09,9E+09,9E+09]],[[184.43,695.20,80.98],[0.0842675,0.873996,0.3985,0.265006],[0,0,0,0],[9E+09,-30,0.00423255,9E+09,9E+09,9E+09]],[[184.43,695.20,80.98],[0.0842675,0.873996,0.3985,0.265006],[0,0,0,0],[9E+09,-30,0.00423255,9E+09,9E+09,9E+09]]],
     [[[184.43,695.20,80.98],[0.0842675,0.873996,0.3985,0.265006],[0,0,0,0],[9E+09,-30,0.00423255,9E+09,9E+09,9E+09]],[[184.43,695.20,80.98],[0.0842675,0.873996,0.3985,0.265006],[0,0,0,0],[9E+09,-30,0.00423255,9E+09,9E+09,9E+09]],[[184.43,695.20,80.98],[0.0842675,0.873996,0.3985,0.265006],[0,0,0,0],[9E+09,-30,0.00423255,9E+09,9E+09,9E+09]]],
     [[[184.43,695.20,80.98],[0.0842675,0.873996,0.3985,0.265006],[0,0,0,0],[9E+09,-30,0.00423255,9E+09,9E+09,9E+09]],[[184.43,695.20,80.98],[0.0842675,0.873996,0.3985,0.265006],[0,0,0,0],[9E+09,-30,0.00423255,9E+09,9E+09,9E+09]],[[184.43,695.20,80.98],[0.0842675,0.873996,0.3985,0.265006],[0,0,0,0],[9E+09,-30,0.00423255,9E+09,9E+09,9E+09]]],
     [[[184.43,695.20,80.98],[0.0842675,0.873996,0.3985,0.265006],[0,0,0,0],[9E+09,-30,0.00423255,9E+09,9E+09,9E+09]],[[184.43,695.20,80.98],[0.0842675,0.873996,0.3985,0.265006],[0,0,0,0],[9E+09,-30,0.00423255,9E+09,9E+09,9E+09]],[[184.43,695.20,80.98],[0.0842675,0.873996,0.3985,0.265006],[0,0,0,0],[9E+09,-30,0.00423255,9E+09,9E+09,9E+09]]],
     [[[184.43,695.20,80.98],[0.0842675,0.873996,0.3985,0.265006],[0,0,0,0],[9E+09,-30,0.00423255,9E+09,9E+09,9E+09]],[[184.43,695.20,80.98],[0.0842675,0.873996,0.3985,0.265006],[0,0,0,0],[9E+09,-30,0.00423255,9E+09,9E+09,9E+09]],[[184.43,695.20,80.98],[0.0842675,0.873996,0.3985,0.265006],[0,0,0,0],[9E+09,-30,0.00423255,9E+09,9E+09,9E+09]]],
     [[[184.43,695.20,80.98],[0.0842675,0.873996,0.3985,0.265006],[0,0,0,0],[9E+09,-30,0.00423255,9E+09,9E+09,9E+09]],[[184.43,695.20,80.98],[0.0842675,0.873996,0.3985,0.265006],[0,0,0,0],[9E+09,-30,0.00423255,9E+09,9E+09,9E+09]],[[184.43,695.20,80.98],[0.0842675,0.873996,0.3985,0.265006],[0,0,0,0],[9E+09,-30,0.00423255,9E+09,9E+09,9E+09]]],
     [[[184.43,695.20,80.98],[0.0842675,0.873996,0.3985,0.265006],[0,0,0,0],[9E+09,-30,0.00423255,9E+09,9E+09,9E+09]],[[184.43,695.20,80.98],[0.0842675,0.873996,0.3985,0.265006],[0,0,0,0],[9E+09,-30,0.00423255,9E+09,9E+09,9E+09]],[[184.43,695.20,80.98],[0.0842675,0.873996,0.3985,0.265006],[0,0,0,0],[9E+09,-30,0.00423255,9E+09,9E+09,9E+09]]],
     [[[184.43,695.20,80.98],[0.0842675,0.873996,0.3985,0.265006],[0,0,0,0],[9E+09,-30,0.00423255,9E+09,9E+09,9E+09]],[[184.43,695.20,80.98],[0.0842675,0.873996,0.3985,0.265006],[0,0,0,0],[9E+09,-30,0.00423255,9E+09,9E+09,9E+09]],[[184.43,695.20,80.98],[0.0842675,0.873996,0.3985,0.265006],[0,0,0,0],[9E+09,-30,0.00423255,9E+09,9E+09,9E+09]]],
     [[[184.43,695.20,80.98],[0.0842675,0.873996,0.3985,0.265006],[0,0,0,0],[9E+09,-30,0.00423255,9E+09,9E+09,9E+09]],[[184.43,695.20,80.98],[0.0842675,0.873996,0.3985,0.265006],[0,0,0,0],[9E+09,-30,0.00423255,9E+09,9E+09,9E+09]],[[184.43,695.20,80.98],[0.0842675,0.873996,0.3985,0.265006],[0,0,0,0],[9E+09,-30,0.00423255,9E+09,9E+09,9E+09]]],
     [[[184.43,695.20,80.98],[0.0842675,0.873996,0.3985,0.265006],[0,0,0,0],[9E+09,-30,0.00423255,9E+09,9E+09,9E+09]],[[184.43,695.20,80.98],[0.0842675,0.873996,0.3985,0.265006],[0,0,0,0],[9E+09,-30,0.00423255,9E+09,9E+09,9E+09]],[[184.43,695.20,80.98],[0.0842675,0.873996,0.3985,0.265006],[0,0,0,0],[9E+09,-30,0.00423255,9E+09,9E+09,9E+09]]],
     [[[184.43,695.20,80.98],[0.0842675,0.873996,0.3985,0.265006],[0,0,0,0],[9E+09,-30,0.00423255,9E+09,9E+09,9E+09]],[[184.43,695.20,80.98],[0.0842675,0.873996,0.3985,0.265006],[0,0,0,0],[9E+09,-30,0.00423255,9E+09,9E+09,9E+09]],[[184.43,695.20,80.98],[0.0842675,0.873996,0.3985,0.265006],[0,0,0,0],[9E+09,-30,0.00423255,9E+09,9E+09,9E+09]]],
     [[[184.43,695.20,80.98],[0.0842675,0.873996,0.3985,0.265006],[0,0,0,0],[9E+09,-30,0.00423255,9E+09,9E+09,9E+09]],[[184.43,695.20,80.98],[0.0842675,0.873996,0.3985,0.265006],[0,0,0,0],[9E+09,-30,0.00423255,9E+09,9E+09,9E+09]],[[184.43,695.20,80.98],[0.0842675,0.873996,0.3985,0.265006],[0,0,0,0],[9E+09,-30,0.00423255,9E+09,9E+09,9E+09]]],
     [[[184.43,695.20,80.98],[0.0842675,0.873996,0.3985,0.265006],[0,0,0,0],[9E+09,-30,0.00423255,9E+09,9E+09,9E+09]],[[184.43,695.20,80.98],[0.0842675,0.873996,0.3985,0.265006],[0,0,0,0],[9E+09,-30,0.00423255,9E+09,9E+09,9E+09]],[[184.43,695.20,80.98],[0.0842675,0.873996,0.3985,0.265006],[0,0,0,0],[9E+09,-30,0.00423255,9E+09,9E+09,9E+09]]],
     [[[184.43,695.20,80.98],[0.0842675,0.873996,0.3985,0.265006],[0,0,0,0],[9E+09,-30,0.00423255,9E+09,9E+09,9E+09]],[[184.43,695.20,80.98],[0.0842675,0.873996,0.3985,0.265006],[0,0,0,0],[9E+09,-30,0.00423255,9E+09,9E+09,9E+09]],[[184.43,695.20,80.98],[0.0842675,0.873996,0.3985,0.265006],[0,0,0,0],[9E+09,-30,0.00423255,9E+09,9E+09,9E+09]]],
     [[[184.43,695.20,80.98],[0.0842675,0.873996,0.3985,0.265006],[0,0,0,0],[9E+09,-30,0.00423255,9E+09,9E+09,9E+09]],[[184.43,695.20,80.98],[0.0842675,0.873996,0.3985,0.265006],[0,0,0,0],[9E+09,-30,0.00423255,9E+09,9E+09,9E+09]],[[184.43,695.20,80.98],[0.0842675,0.873996,0.3985,0.265006],[0,0,0,0],[9E+09,-30,0.00423255,9E+09,9E+09,9E+09]]],
     [[[184.43,695.20,80.98],[0.0842675,0.873996,0.3985,0.265006],[0,0,0,0],[9E+09,-30,0.00423255,9E+09,9E+09,9E+09]],[[184.43,695.20,80.98],[0.0842675,0.873996,0.3985,0.265006],[0,0,0,0],[9E+09,-30,0.00423255,9E+09,9E+09,9E+09]],[[184.43,695.20,80.98],[0.0842675,0.873996,0.3985,0.265006],[0,0,0,0],[9E+09,-30,0.00423255,9E+09,9E+09,9E+09]]],
     [[[184.43,695.20,80.98],[0.0842675,0.873996,0.3985,0.265006],[0,0,0,0],[9E+09,-30,0.00423255,9E+09,9E+09,9E+09]],[[184.43,695.20,80.98],[0.0842675,0.873996,0.3985,0.265006],[0,0,0,0],[9E+09,-30,0.00423255,9E+09,9E+09,9E+09]],[[184.43,695.20,80.98],[0.0842675,0.873996,0.3985,0.265006],[0,0,0,0],[9E+09,-30,0.00423255,9E+09,9E+09,9E+09]]],
     [[[184.43,695.20,80.98],[0.0842675,0.873996,0.3985,0.265006],[0,0,0,0],[9E+09,-30,0.00423255,9E+09,9E+09,9E+09]],[[184.43,695.20,80.98],[0.0842675,0.873996,0.3985,0.265006],[0,0,0,0],[9E+09,-30,0.00423255,9E+09,9E+09,9E+09]],[[184.43,695.20,80.98],[0.0842675,0.873996,0.3985,0.265006],[0,0,0,0],[9E+09,-30,0.00423255,9E+09,9E+09,9E+09]]],
     [[[184.43,695.20,80.98],[0.0842675,0.873996,0.3985,0.265006],[0,0,0,0],[9E+09,-30,0.00423255,9E+09,9E+09,9E+09]],[[184.43,695.20,80.98],[0.0842675,0.873996,0.3985,0.265006],[0,0,0,0],[9E+09,-30,0.00423255,9E+09,9E+09,9E+09]],[[184.43,695.20,80.98],[0.0842675,0.873996,0.3985,0.265006],[0,0,0,0],[9E+09,-30,0.00423255,9E+09,9E+09,9E+09]]],
     [[[184.43,695.20,80.98],[0.0842675,0.873996,0.3985,0.265006],[0,0,0,0],[9E+09,-30,0.00423255,9E+09,9E+09,9E+09]],[[184.43,695.20,80.98],[0.0842675,0.873996,0.3985,0.265006],[0,0,0,0],[9E+09,-30,0.00423255,9E+09,9E+09,9E+09]],[[184.43,695.20,80.98],[0.0842675,0.873996,0.3985,0.265006],[0,0,0,0],[9E+09,-30,0.00423255,9E+09,9E+09,9E+09]]],
     [[[184.43,695.20,80.98],[0.0842675,0.873996,0.3985,0.265006],[0,0,0,0],[9E+09,-30,0.00423255,9E+09,9E+09,9E+09]],[[184.43,695.20,80.98],[0.0842675,0.873996,0.3985,0.265006],[0,0,0,0],[9E+09,-30,0.00423255,9E+09,9E+09,9E+09]],[[184.43,695.20,80.98],[0.0842675,0.873996,0.3985,0.265006],[0,0,0,0],[9E+09,-30,0.00423255,9E+09,9E+09,9E+09]]],
     [[[184.43,695.20,80.98],[0.0842675,0.873996,0.3985,0.265006],[0,0,0,0],[9E+09,-30,0.00423255,9E+09,9E+09,9E+09]],[[184.43,695.20,80.98],[0.0842675,0.873996,0.3985,0.265006],[0,0,0,0],[9E+09,-30,0.00423255,9E+09,9E+09,9E+09]],[[184.43,695.20,80.98],[0.0842675,0.873996,0.3985,0.265006],[0,0,0,0],[9E+09,-30,0.00423255,9E+09,9E+09,9E+09]]],
     [[[184.43,695.20,80.98],[0.0842675,0.873996,0.3985,0.265006],[0,0,0,0],[9E+09,-30,0.00423255,9E+09,9E+09,9E+09]],[[184.43,695.20,80.98],[0.0842675,0.873996,0.3985,0.265006],[0,0,0,0],[9E+09,-30,0.00423255,9E+09,9E+09,9E+09]],[[184.43,695.20,80.98],[0.0842675,0.873996,0.3985,0.265006],[0,0,0,0],[9E+09,-30,0.00423255,9E+09,9E+09,9E+09]]],
     [[[184.43,695.20,80.98],[0.0842675,0.873996,0.3985,0.265006],[0,0,0,0],[9E+09,-30,0.00423255,9E+09,9E+09,9E+09]],[[184.43,695.20,80.98],[0.0842675,0.873996,0.3985,0.265006],[0,0,0,0],[9E+09,-30,0.00423255,9E+09,9E+09,9E+09]],[[184.43,695.20,80.98],[0.0842675,0.873996,0.3985,0.265006],[0,0,0,0],[9E+09,-30,0.00423255,9E+09,9E+09,9E+09]]],
	 [[[184.43,695.20,80.98],[0.0842675,0.873996,0.3985,0.265006],[0,0,0,0],[9E+09,-30,0.00423255,9E+09,9E+09,9E+09]],[[184.43,695.20,80.98],[0.0842675,0.873996,0.3985,0.265006],[0,0,0,0],[9E+09,-30,0.00423255,9E+09,9E+09,9E+09]],[[184.43,695.20,80.98],[0.0842675,0.873996,0.3985,0.265006],[0,0,0,0],[9E+09,-30,0.00423255,9E+09,9E+09,9E+09]]],
     [[[184.43,695.20,80.98],[0.0842675,0.873996,0.3985,0.265006],[0,0,0,0],[9E+09,-30,0.00423255,9E+09,9E+09,9E+09]],[[184.43,695.20,80.98],[0.0842675,0.873996,0.3985,0.265006],[0,0,0,0],[9E+09,-30,0.00423255,9E+09,9E+09,9E+09]],[[184.43,695.20,80.98],[0.0842675,0.873996,0.3985,0.265006],[0,0,0,0],[9E+09,-30,0.00423255,9E+09,9E+09,9E+09]]],
     [[[184.43,695.20,80.98],[0.0842675,0.873996,0.3985,0.265006],[0,0,0,0],[9E+09,-30,0.00423255,9E+09,9E+09,9E+09]],[[184.43,695.20,80.98],[0.0842675,0.873996,0.3985,0.265006],[0,0,0,0],[9E+09,-30,0.00423255,9E+09,9E+09,9E+09]],[[184.43,695.20,80.98],[0.0842675,0.873996,0.3985,0.265006],[0,0,0,0],[9E+09,-30,0.00423255,9E+09,9E+09,9E+09]]],
     [[[184.43,695.20,80.98],[0.0842675,0.873996,0.3985,0.265006],[0,0,0,0],[9E+09,-30,0.00423255,9E+09,9E+09,9E+09]],[[184.43,695.20,80.98],[0.0842675,0.873996,0.3985,0.265006],[0,0,0,0],[9E+09,-30,0.00423255,9E+09,9E+09,9E+09]],[[184.43,695.20,80.98],[0.0842675,0.873996,0.3985,0.265006],[0,0,0,0],[9E+09,-30,0.00423255,9E+09,9E+09,9E+09]]],
     [[[184.43,695.20,80.98],[0.0842675,0.873996,0.3985,0.265006],[0,0,0,0],[9E+09,-30,0.00423255,9E+09,9E+09,9E+09]],[[184.43,695.20,80.98],[0.0842675,0.873996,0.3985,0.265006],[0,0,0,0],[9E+09,-30,0.00423255,9E+09,9E+09,9E+09]],[[184.43,695.20,80.98],[0.0842675,0.873996,0.3985,0.265006],[0,0,0,0],[9E+09,-30,0.00423255,9E+09,9E+09,9E+09]]],
     [[[184.43,695.20,80.98],[0.0842675,0.873996,0.3985,0.265006],[0,0,0,0],[9E+09,-30,0.00423255,9E+09,9E+09,9E+09]],[[184.43,695.20,80.98],[0.0842675,0.873996,0.3985,0.265006],[0,0,0,0],[9E+09,-30,0.00423255,9E+09,9E+09,9E+09]],[[184.43,695.20,80.98],[0.0842675,0.873996,0.3985,0.265006],[0,0,0,0],[9E+09,-30,0.00423255,9E+09,9E+09,9E+09]]],
     [[[184.43,695.20,80.98],[0.0842675,0.873996,0.3985,0.265006],[0,0,0,0],[9E+09,-30,0.00423255,9E+09,9E+09,9E+09]],[[184.43,695.20,80.98],[0.0842675,0.873996,0.3985,0.265006],[0,0,0,0],[9E+09,-30,0.00423255,9E+09,9E+09,9E+09]],[[184.43,695.20,80.98],[0.0842675,0.873996,0.3985,0.265006],[0,0,0,0],[9E+09,-30,0.00423255,9E+09,9E+09,9E+09]]],
     [[[184.43,695.20,80.98],[0.0842675,0.873996,0.3985,0.265006],[0,0,0,0],[9E+09,-30,0.00423255,9E+09,9E+09,9E+09]],[[184.43,695.20,80.98],[0.0842675,0.873996,0.3985,0.265006],[0,0,0,0],[9E+09,-30,0.00423255,9E+09,9E+09,9E+09]],[[184.43,695.20,80.98],[0.0842675,0.873996,0.3985,0.265006],[0,0,0,0],[9E+09,-30,0.00423255,9E+09,9E+09,9E+09]]],
     [[[184.43,695.20,80.98],[0.0842675,0.873996,0.3985,0.265006],[0,0,0,0],[9E+09,-30,0.00423255,9E+09,9E+09,9E+09]],[[184.43,695.20,80.98],[0.0842675,0.873996,0.3985,0.265006],[0,0,0,0],[9E+09,-30,0.00423255,9E+09,9E+09,9E+09]],[[184.43,695.20,80.98],[0.0842675,0.873996,0.3985,0.265006],[0,0,0,0],[9E+09,-30,0.00423255,9E+09,9E+09,9E+09]]],
     [[[184.43,695.20,80.98],[0.0842675,0.873996,0.3985,0.265006],[0,0,0,0],[9E+09,-30,0.00423255,9E+09,9E+09,9E+09]],[[184.43,695.20,80.98],[0.0842675,0.873996,0.3985,0.265006],[0,0,0,0],[9E+09,-30,0.00423255,9E+09,9E+09,9E+09]],[[184.43,695.20,80.98],[0.0842675,0.873996,0.3985,0.265006],[0,0,0,0],[9E+09,-30,0.00423255,9E+09,9E+09,9E+09]]]];

! ChanLam and Chan searches

PERS robtarget LL_ChanLam_Xs:=[[-315,167.5,36.707],[5.66804E-07,-0.719939,-0.694038,8.58113E-08],[0,1,-3,0],[9E+09,-45,0.00398376,9E+09,9E+09,9E+09]];
PERS robtarget LL_ChanLam_Xe:=[[-275,167.5,36.707],[1.64071E-07,-0.719937,-0.69404,4.08933E-07],[0,1,-3,0],[9E+09,-45,0.00398376,9E+09,9E+09,9E+09]];
PERS robtarget LL_Chan_Xs:=[[-309,757.5,36.707],[2.23894E-07,-0.719937,-0.69404,4.99141E-07],[0,1,-3,0],[9E+09,-45,0.00394822,9E+09,9E+09,9E+09]];
PERS robtarget LL_Chan_Xe:=[[-269,757.5,36.707],[5.56529E-07,0.719937,0.69404,1.1896E-06],[0,1,-3,0],[9E+09,-45,0.00398376,9E+09,9E+09,9E+09]];

PERS robtarget RL_ChanLam_Xs:=[[315,167.5,39.262],[2.58776E-06,-0.719939,-0.694037,1.11975E-08],[0,1,-3,0],[9E+09,-45,0.00398376,9E+09,9E+09,9E+09]];
PERS robtarget RL_ChanLam_Xe:=[[275,167.5,39.262],[1.85214E-06,-0.719938,-0.694039,7.39728E-07],[0,1,-3,0],[9E+09,-45,0.00398376,9E+09,9E+09,9E+09]];
PERS robtarget RL_Chan_Xs:=[[309,757.5,41.1448],[4.05915E-07,0.719938,0.694038,-1.35012E-06],[0,1,-3,0],[9E+09,-45,0.00398376,9E+09,9E+09,9E+09]];
PERS robtarget RL_Chan_Xe:=[[269,757.5,41.1448],[1.31705E-06,-0.719939,-0.694038,-6.77001E-07],[0,1,-3,0],[9E+09,-45,0.00394822,9E+09,9E+09,9E+09]];

PERS robtarget RR_ChanLam_Xs:=[[315,167.5,39.9118],[6.01662E-07,0.588726,-0.808333,-6.35659E-07],[-1,1,-2,0],[9E+09,-44.0856,180,9E+09,9E+09,9E+09]];
PERS robtarget RR_ChanLam_Xe:=[[275,167.5,39.9118],[2.60299E-07,0.588723,-0.808335,3.43015E-07],[-1,1,-2,0],[9E+09,-44.0856,180,9E+09,9E+09,9E+09]];
PERS robtarget RR_Chan_Xs:=[[309,757.5,39.1934],[2.36753E-07,-0.588727,0.808332,5.26239E-07],[-1,1,-2,0],[9E+09,-44.0856,180,9E+09,9E+09,9E+09]];
PERS robtarget RR_Chan_Xe:=[[269,757.5,39.1934],[9.04661E-07,0.588725,-0.808333,-2.14368E-07],[-1,1,-2,0],[9E+09,-44.0856,180,9E+09,9E+09,9E+09]];

PERS robtarget LR_ChanLam_Xs:=[[-315,167.5,41.7754],[2.52881E-07,0.588726,-0.808333,-1.78206E-07],[-1,1,-2,0],[9E+09,-44.0856,180,9E+09,9E+09,9E+09]];
PERS robtarget LR_ChanLam_Xe:=[[-275,167.5,41.7754],[2.91328E-07,0.588725,-0.808333,-5.94468E-07],[-1,1,-2,0],[9E+09,-44.0856,180,9E+09,9E+09,9E+09]];
PERS robtarget LR_Chan_Xs:=[[-309,757.5,41.0798],[2.22579E-05,-0.588712,0.808343,-6.78295E-05],[-1,1,-3,0],[9E+09,-44.0856,180,9E+09,9E+09,9E+09]];
PERS robtarget LR_Chan_Xe:=[[-269,757.5,41.0798],[2.14432E-05,-0.58871,0.808345,-6.79108E-05],[-1,1,-3,0],[9E+09,-44.0856,180,9E+09,9E+09,9E+09]];

PERS robtarget LL_ChanLam_Zs:=[[-309,167.5,109.5],[0.672196,-0.219437,-0.672197,0.219435],[0,1,-4,0],[9E+09,-45,0.00385937,9E+09,9E+09,9E+09]];
PERS robtarget LL_ChanLam_Ze:=[[-309,167.5,69.5],[0.672196,-0.219433,-0.672198,0.219437],[0,1,-4,0],[9E+09,-45,0.00385937,9E+09,9E+09,9E+09]];
PERS robtarget LL_Chan_Zs:=[[-309,757.5,109.5],[0.672196,-0.219434,-0.672197,0.219436],[0,1,-4,0],[9E+09,-45,0.00385937,9E+09,9E+09,9E+09]];
PERS robtarget LL_Chan_Ze:=[[-309,757.5,69.5],[0.672195,-0.219436,-0.672198,0.219436],[0,1,-4,0],[9E+09,-45,0.00385937,9E+09,9E+09,9E+09]];

PERS robtarget RL_ChanLam_Zs:=[[309,167.5,109.5],[0.184899,0.682505,0.1849,0.682504],[0,0,-1,0],[9E+09,-43.169,-1.8285,9E+09,9E+09,9E+09]];
PERS robtarget RL_ChanLam_Ze:=[[309,167.5,69.5],[0.184898,0.682507,0.184898,0.682503],[0,0,-1,0],[9E+09,-43.1689,-1.8285,9E+09,9E+09,9E+09]];
PERS robtarget RL_Chan_Zs:=[[309,757.5,109.5],[0.184898,0.682507,0.184899,0.682502],[0,0,-1,0],[9E+09,-43.1689,-1.8285,9E+09,9E+09,9E+09]];
PERS robtarget RL_Chan_Ze:=[[309,757.5,69.5],[0.184898,0.682506,0.184898,0.682504],[0,0,-1,0],[9E+09,-43.1689,-1.82854,9E+09,9E+09,9E+09]];

PERS robtarget RR_ChanLam_Zs:=[[309,167.5,109.5],[0.183528,-0.682873,0.183528,-0.682876],[-1,1,0,0],[9E+09,-45,180,9E+09,9E+09,9E+09]];
PERS robtarget RR_ChanLam_Ze:=[[309,167.5,69.5],[0.18353,-0.682873,0.183527,-0.682876],[-1,1,0,0],[9E+09,-45,180,9E+09,9E+09,9E+09]];
PERS robtarget RR_Chan_Zs:=[[309,757.5,109.5],[0.183545,-0.682889,0.183518,-0.682858],[-1,1,0,0],[9E+09,-45.0001,180,9E+09,9E+09,9E+09]];
PERS robtarget RR_Chan_Ze:=[[309,757.5,69.5],[0.183546,-0.682889,0.183519,-0.682858],[-1,1,0,0],[9E+09,-45.0001,180,9E+09,9E+09,9E+09]];

PERS robtarget LR_ChanLam_Zs:=[[-309,167.5,109.5],[0.703916,0.0670874,-0.703918,-0.067087],[-1,0,-1,0],[9E+09,-45,180,9E+09,9E+09,9E+09]];
PERS robtarget LR_ChanLam_Ze:=[[-309,167.5,69.5],[0.703917,0.0670859,-0.703917,-0.0670864],[-1,0,-1,0],[9E+09,-45,180,9E+09,9E+09,9E+09]];
PERS robtarget LR_Chan_Zs:=[[-309,757.5,109.5],[0.703917,0.0670848,-0.703917,-0.0670882],[-1,0,-1,0],[9E+09,-45,180,9E+09,9E+09,9E+09]];
PERS robtarget LR_Chan_Ze:=[[-309,757.5,69.5],[0.703917,0.0670878,-0.703917,-0.067088],[-1,0,-1,0],[9E+09,-45,180,9E+09,9E+09,9E+09]];

PERS robtarget Found_ChanLam_X:=[[-274.721,167.511,41.7626],[2.71318E-05,-0.588733,0.808327,-3.01854E-05],[-1,1,-2,0],[9E+09,-44.0856,180,9E+09,9E+09,9E+09]];
PERS robtarget Found_Chan_X:=[[-272.124,757.5,41.0922],[2.80223E-05,-0.588695,0.808355,-5.46964E-05],[-1,1,-3,0],[9E+09,-44.0856,180,9E+09,9E+09,9E+09]];


PROC Plan_Duh_Chan()


    ALL_Chan_Plan 50;
    WaitTime\InPos,.2;
    LLnRR_CHAN_PLAN Horiz_Y1;
    WaitTime\InPos,.2;
    LLnRR_CHAN_PLAN Horiz_Y2;
    WaitTime\InPos,.2;
    LLnRR_CHAN_PLAN Horiz_Y3;
    WaitTime\InPos,.2;
    LLnRR_CHAN_PLAN Horiz_Y4;
    WaitTime\InPos,.2;
    LRnRL_CHAN_PLAN "Anchor";
    WaitTime\InPos,.2;
    LRnRL_CHAN_PLAN "Push_Stop";
    WaitTime\InPos,.2;
    LRnRL_CHAN_PLAN "Chan_Bottom";
    WaitTime\InPos,.2;
    LRnRL_CHAN_PLAN "Y3";
    WaitTime\InPos,.2;
    LRnRL_CHAN_PLAN "Y4";
    WaitTime\InPos,.2;


FOR z FROM 2 TO How_Many
STEP + 1 DO
 ! added 7/10/20/SS
	! if TIGHTBOX = TRUE then skip everything above it...
	! this may have a flaw, if there is a tight box in the middle of the part and not a TIGHTBOX above it..
	! but I have never seen one like that before.

IF (LR_CHAN_WELDS{z,1}.trans.Y > HORIZ_Y3 or LR_CHAN_WELDS{z,2}.trans.Y > HORIZ_Y3 or LR_CHAN_WELDS{z,3}.trans.Y > HORIZ_Y3) AND Y3_TightBox = TRUE  THEN
		    LR_CHAN_NOTES{z,1} := "SKIP";
			RL_CHAN_NOTES{z,1} := "SKIP";
ENDIF

IF  RL_CHAN_WELDS{z,1}.trans.Y > HORIZ_Y4 AND Y4_TightBox = TRUE  THEN
		    LR_CHAN_NOTES{z,1} := "SKIP";
			RL_CHAN_NOTES{z,1} := "SKIP";
ENDIF
ENDFOR


ENDPROC



PROC ALL_OF_THE_CHANNELS()

    SET_CHAN_SEARCHES;
    ActUnit STN1;
    Plan_Duh_Chan;
    WELD_LL_CHANNEL;
    WELD_RL_CHANNEL;
    WELD_RR_CHANNEL;
    WELD_LR_CHANNEL;
    This_Channel_Sucks:

ENDPROC

    PROC SET_CHAN_SEARCHES()


        !!!@@@@@@@@@@@@@@@@@@@@@@@
        LL_ChanLam_Xs.TRANS.X := LX2 - NOZZLE_RADIUS - SEARCH_LENGTH;
        LL_ChanLam_Xe.TRANS.X := LX2 - NOZZLE_RADIUS;
        LL_Chan_Xs.TRANS.X := LX2 + BAR_THICKNESS - NOZZLE_RADIUS - SEARCH_LENGTH;
        LL_Chan_Xe.TRANS.X := LX2 + BAR_THICKNESS - NOZZLE_RADIUS;
        !!!!!!!!!!@
        LR_ChanLam_Xs.TRANS.X := LX2 - NOZZLE_RADIUS - SEARCH_LENGTH;
        LR_ChanLam_Xe.TRANS.X := LX2 - NOZZLE_RADIUS;
        LR_Chan_Xs.TRANS.X := LX2 + BAR_THICKNESS - NOZZLE_RADIUS - SEARCH_LENGTH;
        LR_Chan_Xe.TRANS.X := LX2 + BAR_THICKNESS - NOZZLE_RADIUS;

        !!!!!!!!!!#
        RR_ChanLam_Xs.TRANS.X := RX2 + NOZZLE_RADIUS + SEARCH_LENGTH;
        RR_ChanLam_Xe.TRANS.X := RX2 + NOZZLE_RADIUS;
        RR_Chan_Xs.TRANS.X := RX2 - BAR_THICKNESS + NOZZLE_RADIUS + SEARCH_LENGTH;
        RR_Chan_Xe.TRANS.X := RX2 - BAR_THICKNESS + NOZZLE_RADIUS;

        RL_ChanLam_Xs.TRANS.X := RX2 + NOZZLE_RADIUS + SEARCH_LENGTH;
        RL_ChanLam_Xe.TRANS.X := RX2 + NOZZLE_RADIUS;
        RL_Chan_Xs.TRANS.X := RX2 - BAR_THICKNESS + NOZZLE_RADIUS + SEARCH_LENGTH;
        RL_Chan_Xe.TRANS.X := RX2 - BAR_THICKNESS + NOZZLE_RADIUS;


        LL_ChanLam_Zs.TRANS.X := LX2 - (NOZZLE_LENGTH/2);
        LL_ChanLam_Ze.TRANS.X :=  LX2 - (NOZZLE_LENGTH/2);
        LL_Chan_Zs.TRANS.X :=  LX2 - (NOZZLE_LENGTH/2);
        LL_Chan_Ze.TRANS.X :=  LX2 - (NOZZLE_LENGTH/2);
        !!!!!!!!!!@
        LR_ChanLam_Zs.TRANS.X :=  LX2 - (NOZZLE_LENGTH/2);
        LR_ChanLam_Ze.TRANS.X :=  LX2 - (NOZZLE_LENGTH/2);
        LR_Chan_Zs.TRANS.X :=  LX2 - (NOZZLE_LENGTH/2);
        LR_Chan_Ze.TRANS.X :=  LX2 - (NOZZLE_LENGTH/2);

        !!!!!!!!!!#
        RR_ChanLam_Zs.TRANS.X := RX2 + (NOZZLE_LENGTH/2);
        RR_ChanLam_Ze.TRANS.X := RX2 + (NOZZLE_LENGTH/2);
        RR_Chan_Zs.TRANS.X := RX2 + (NOZZLE_LENGTH/2);
        RR_Chan_Ze.TRANS.X :=  RX2 + (NOZZLE_LENGTH/2);

        RL_ChanLam_Zs.TRANS.X := RX2 + (NOZZLE_LENGTH/2);
        RL_ChanLam_Ze.TRANS.X := RX2 + (NOZZLE_LENGTH/2);
        RL_Chan_Zs.TRANS.X := RX2 + (NOZZLE_LENGTH/2);
        RL_Chan_Ze.TRANS.X := RX2 + (NOZZLE_LENGTH/2);

        LL_ChanLam_Zs.TRANS.Z := TOP_O_BARZ + SEARCH_LENGTH;
        LL_ChanLam_Ze.TRANS.Z := TOP_O_BARZ ;
        LL_Chan_Zs.TRANS.Z := TOP_O_BARZ + SEARCH_LENGTH;
        LL_Chan_Ze.TRANS.Z := TOP_O_BARZ ;

        LR_ChanLam_Zs.TRANS.Z := TOP_O_BARZ + SEARCH_LENGTH;
        LR_ChanLam_Ze.TRANS.Z := TOP_O_BARZ ;
        LR_Chan_Zs.TRANS.Z := TOP_O_BARZ  + SEARCH_LENGTH;
        LR_Chan_Ze.TRANS.Z := TOP_O_BARZ ;

        RR_ChanLam_Zs.TRANS.Z := TOP_O_BARZ + SEARCH_LENGTH;
        RR_ChanLam_Ze.TRANS.Z := TOP_O_BARZ ;
        RR_Chan_Zs.TRANS.Z := TOP_O_BARZ  + SEARCH_LENGTH;
        RR_Chan_Ze.TRANS.Z := TOP_O_BARZ ;

        RL_ChanLam_Zs.TRANS.Z := TOP_O_BARZ + SEARCH_LENGTH;
        RL_ChanLam_Ze.TRANS.Z := TOP_O_BARZ ;
        RL_Chan_Zs.TRANS.Z := TOP_O_BARZ + SEARCH_LENGTH;
        RL_Chan_Ze.TRANS.Z :=TOP_O_BARZ ;

           IF LOAD_PUSH = FALSE THEN

        LL_ChanLam_Xs.TRANS.Y := HORIZ_Y2 + BAR_THICKNESS + NOZZLE_RADIUS + SEARCH_LENGTH;
        LL_ChanLam_Xe.TRANS.Y := HORIZ_Y2 + BAR_THICKNESS + NOZZLE_RADIUS + SEARCH_LENGTH;
        LL_Chan_Xs.TRANS.Y := Top_Of_Chan_Y - ( CHANNEL_LENGTH/2);
        LL_Chan_Xe.TRANS.Y := Top_Of_Chan_Y - ( CHANNEL_LENGTH/2);

        LR_ChanLam_Xs.TRANS.Y := HORIZ_Y2 + BAR_THICKNESS + NOZZLE_RADIUS + SEARCH_LENGTH;
        LR_ChanLam_Xe.TRANS.Y := HORIZ_Y2 + BAR_THICKNESS + NOZZLE_RADIUS + SEARCH_LENGTH;
        LR_Chan_Xs.TRANS.Y := Top_Of_Chan_Y - ( CHANNEL_LENGTH/2);
        LR_Chan_Xe.TRANS.Y := Top_Of_Chan_Y - ( CHANNEL_LENGTH/2);

        RR_ChanLam_Xs.TRANS.Y := HORIZ_Y2 + BAR_THICKNESS + NOZZLE_RADIUS + SEARCH_LENGTH;
        RR_ChanLam_Xe.TRANS.Y := HORIZ_Y2 + BAR_THICKNESS + NOZZLE_RADIUS + SEARCH_LENGTH;
        RR_Chan_Xs.TRANS.Y := Top_Of_Chan_Y - ( CHANNEL_LENGTH/2);
        RR_Chan_Xe.TRANS.Y := Top_Of_Chan_Y - ( CHANNEL_LENGTH/2);

        RL_ChanLam_Xs.TRANS.Y := HORIZ_Y2 + BAR_THICKNESS + NOZZLE_RADIUS + SEARCH_LENGTH;
        RL_ChanLam_Xe.TRANS.Y := HORIZ_Y2 + BAR_THICKNESS + NOZZLE_RADIUS + SEARCH_LENGTH;
        RL_Chan_Xs.TRANS.Y := Top_Of_Chan_Y - ( CHANNEL_LENGTH/2);
        RL_Chan_Xe.TRANS.Y := Top_Of_Chan_Y - ( CHANNEL_LENGTH/2);


        LL_ChanLam_Zs.TRANS.Y := HORIZ_Y2 + BAR_THICKNESS + NOZZLE_RADIUS + SEARCH_LENGTH;
        LL_ChanLam_Ze.TRANS.Y := HORIZ_Y2 + BAR_THICKNESS + NOZZLE_RADIUS + SEARCH_LENGTH;
        LL_Chan_Zs.TRANS.Y := Top_Of_Chan_Y - ( CHANNEL_LENGTH/2);
        LL_Chan_Ze.TRANS.Y := Top_Of_Chan_Y - ( CHANNEL_LENGTH/2);

        LR_ChanLam_Zs.TRANS.Y := HORIZ_Y2 + BAR_THICKNESS + NOZZLE_RADIUS + SEARCH_LENGTH;
        LR_ChanLam_Ze.TRANS.Y := HORIZ_Y2 + BAR_THICKNESS + NOZZLE_RADIUS + SEARCH_LENGTH;
        LR_Chan_Zs.TRANS.Y := Top_Of_Chan_Y - ( CHANNEL_LENGTH/2);
        LR_Chan_Ze.TRANS.Y := Top_Of_Chan_Y - ( CHANNEL_LENGTH/2);

        RR_ChanLam_Zs.TRANS.Y := HORIZ_Y2 + BAR_THICKNESS + NOZZLE_RADIUS + SEARCH_LENGTH;
        RR_ChanLam_Ze.TRANS.Y := HORIZ_Y2 + BAR_THICKNESS + NOZZLE_RADIUS + SEARCH_LENGTH;
        RR_Chan_Zs.TRANS.Y := Top_Of_Chan_Y - ( CHANNEL_LENGTH/2);
        RR_Chan_Ze.TRANS.Y := Top_Of_Chan_Y - ( CHANNEL_LENGTH/2);

        RL_ChanLam_Zs.TRANS.Y := HORIZ_Y2 + BAR_THICKNESS + NOZZLE_RADIUS + SEARCH_LENGTH;
        RL_ChanLam_Ze.TRANS.Y := HORIZ_Y2 + BAR_THICKNESS + NOZZLE_RADIUS + SEARCH_LENGTH;
        RL_Chan_Zs.TRANS.Y := Top_Of_Chan_Y - ( CHANNEL_LENGTH/2);
        RL_Chan_Ze.TRANS.Y := Top_Of_Chan_Y - ( CHANNEL_LENGTH/2);


        ELSEIF LOAD_PUSH = TRUE THEN

        LL_ChanLam_Xs.TRANS.Y :=  HORIZ_Y1 + BAR_THICKNESS + NOZZLE_RADIUS + SEARCH_LENGTH;
        LL_ChanLam_Xe.TRANS.Y :=  HORIZ_Y1 + BAR_THICKNESS + NOZZLE_RADIUS + SEARCH_LENGTH;
        LL_Chan_Xs.TRANS.Y := Top_Of_Chan_Y - ( CHANNEL_LENGTH/2);
        LL_Chan_Xe.TRANS.Y := Top_Of_Chan_Y - ( CHANNEL_LENGTH/2);

        RR_ChanLam_Xs.TRANS.Y :=  HORIZ_Y1 + BAR_THICKNESS + NOZZLE_RADIUS + SEARCH_LENGTH;
        RR_ChanLam_Xe.TRANS.Y :=  HORIZ_Y1 + BAR_THICKNESS + NOZZLE_RADIUS + SEARCH_LENGTH;
        RR_Chan_Xs.TRANS.Y := Top_Of_Chan_Y - ( CHANNEL_LENGTH/2);
        RR_Chan_Xe.TRANS.Y := Top_Of_Chan_Y - ( CHANNEL_LENGTH/2);

        LR_ChanLam_Xs.TRANS.Y :=  HORIZ_Y1 + BAR_THICKNESS + NOZZLE_RADIUS + SEARCH_LENGTH;
        LR_ChanLam_Xe.TRANS.Y :=  HORIZ_Y1 + BAR_THICKNESS + NOZZLE_RADIUS + SEARCH_LENGTH;
        LR_Chan_Xs.TRANS.Y := Top_Of_Chan_Y - ( CHANNEL_LENGTH/2);
        LR_Chan_Xe.TRANS.Y := Top_Of_Chan_Y - ( CHANNEL_LENGTH/2);

        RL_ChanLam_Xs.TRANS.Y :=  HORIZ_Y1 + BAR_THICKNESS + NOZZLE_RADIUS + SEARCH_LENGTH;
        RL_ChanLam_Xe.TRANS.Y :=  HORIZ_Y1 + BAR_THICKNESS + NOZZLE_RADIUS + SEARCH_LENGTH;
        RL_Chan_Xs.TRANS.Y := Top_Of_Chan_Y - ( CHANNEL_LENGTH/2);
        RL_Chan_Xe.TRANS.Y := Top_Of_Chan_Y - ( CHANNEL_LENGTH/2);


        LL_ChanLam_Zs.TRANS.Y :=  HORIZ_Y1 + BAR_THICKNESS + NOZZLE_RADIUS + SEARCH_LENGTH;
        LL_ChanLam_Ze.TRANS.Y :=  HORIZ_Y1 + BAR_THICKNESS + NOZZLE_RADIUS + SEARCH_LENGTH;
        LL_Chan_Zs.TRANS.Y := Top_Of_Chan_Y - ( CHANNEL_LENGTH/2);
        LL_Chan_Ze.TRANS.Y := Top_Of_Chan_Y - ( CHANNEL_LENGTH/2);

        RR_ChanLam_Zs.TRANS.Y :=  HORIZ_Y1 + BAR_THICKNESS + NOZZLE_RADIUS + SEARCH_LENGTH;
        RR_ChanLam_Ze.TRANS.Y :=  HORIZ_Y1 + BAR_THICKNESS + NOZZLE_RADIUS + SEARCH_LENGTH;
        RR_Chan_Zs.TRANS.Y := Top_Of_Chan_Y - ( CHANNEL_LENGTH/2);
        RR_Chan_Ze.TRANS.Y := Top_Of_Chan_Y - ( CHANNEL_LENGTH/2);

        LR_ChanLam_Zs.TRANS.Y :=  HORIZ_Y1 + BAR_THICKNESS + NOZZLE_RADIUS + SEARCH_LENGTH;
        LR_ChanLam_Ze.TRANS.Y :=  HORIZ_Y1 + BAR_THICKNESS + NOZZLE_RADIUS + SEARCH_LENGTH;
        LR_Chan_Zs.TRANS.Y := Top_Of_Chan_Y - ( CHANNEL_LENGTH/2);
        LR_Chan_Ze.TRANS.Y := Top_Of_Chan_Y - ( CHANNEL_LENGTH/2);

        RL_ChanLam_Zs.TRANS.Y :=  HORIZ_Y1 + BAR_THICKNESS + NOZZLE_RADIUS + SEARCH_LENGTH;
        RL_ChanLam_Ze.TRANS.Y :=  HORIZ_Y1 + BAR_THICKNESS + NOZZLE_RADIUS + SEARCH_LENGTH;
        RL_Chan_Zs.TRANS.Y := Top_Of_Chan_Y - ( CHANNEL_LENGTH/2);
        RL_Chan_Ze.TRANS.Y := Top_Of_Chan_Y - ( CHANNEL_LENGTH/2);

        ENDIF
        WAITTIME\INPOS, 1;

        ENDPROC


    PROC WELD_LL_CHANNEL()

    ActUnit Stn1;
    AccSet 100, STOP_DA_SLOP;
    PDispOff;

    MoveJ [[-262.03,450.00,360.03],[0.0589426,0.939499,0.2242,0.252193],[0,1,-2,0],[9E+09,-25,0.00394822,9E+09,9E+09,9E+09]], V500, Z100, tWeldGun\WObj:=WobJ_FacePlates;

    MoveJ OFFS(LL_ChanLam_Zs,0,0,250),v1000,Z100,tWeldGun\WObj:=WobJ_FacePlates;
    MoveL Offs(LL_ChanLam_Zs,0,0,50),v1000,Z100,tWeldGun\WObj:=WobJ_FacePlates;

    Search_1D SR_ChanLam_FOUND\SearchStop:=CHANLAM_Found_Z, LL_ChanLam_Zs, LL_ChanLam_Ze, V200, tWeldGun\WObj:=WobJ_FacePlates\SchSpeed:=15;
    XnY_Depth LL_ChanLam_Xs, LL_ChanLam_Xe, Found_Z, 23;

    MoveL Offs(LL_ChanLam_Zs,0,0,100),v1000,Z100,tWeldGun\WObj:=WobJ_FacePlates;
    MoveL Offs(LL_Chan_Zs,0,0,100),v1000,Z100,tWeldGun\WObj:=WobJ_FacePlates;

    Search_1D SR_Chan_FOUND\SearchStop:=CHAN_Found_Z, LL_Chan_Zs, LL_Chan_Ze, V200, tWeldGun\WObj:=WobJ_FacePlates\SchSpeed:=15;
    XnY_Depth LL_Chan_Xs, LL_Chan_Xe, Found_Z, 23;
    SET_CHAN_Zs "LL";

    MoveL Offs(LL_Chan_Zs,0,0,250),v1000,Z100,tWeldGun\WObj:=WobJ_FacePlates;
    MoveJ Offs(LL_ChanLam_Xs,0,0,150),v1000,Z100,tWeldGun\WObj:=WobJ_FacePlates;
    MoveL RelTooL(LL_ChanLam_Xs,0,0,-75),v1000,Z100,tWeldGun\WObj:=WobJ_FacePlates;

    Search_1D SR_ChanLam_FOUND\SearchStop:=Found_ChanLam_X, LL_ChanLam_Xs, LL_ChanLam_Xe, V200, tWeldGun\WObj:=WobJ_FacePlates\SchSpeed:=15;

    MoveL RelTooL(LL_ChanLam_Xs,0,0,-100),v1000,Z100,tWeldGun\WObj:=WobJ_FacePlates;
    MoveL RelTooL(LL_Chan_Xs,0,0,-100),v1000,Z100,tWeldGun\WObj:=WobJ_FacePlates;

    Search_1D SR_Chan_FOUND\SearchStop:=Found_Chan_X, LL_Chan_Xs, LL_Chan_Xe, V200, tWeldGun\WObj:=WobJ_FacePlates\SchSpeed:=15;

    MoveL RelTooL(LL_Chan_Xs,0,0,-150),v1000,Z100,tWeldGun\WObj:=WobJ_FacePlates;
    PDispOff;

    SET_LL_ChanX;


  IF WeldEVENs_Outside_LLnRR = TRUE THEN
    FOR w FROM 2 TO How_Many
     STEP +2 DO
        GENERIC_LL_STITCH w;
           IF w+2 > How_Many THEN
           BACK_AWAY 450;
               ! MoveL Offs(LL_CHAN_WELDS{w,1},0,0,250),V500,Z10,tWeldGun\WObj:=WobJ_FacePlates;
           ENDIF
    ENDFOR

  ELSEIF WeldEVENs_Outside_LLnRR = FALSE THEN
    FOR w FROM 1 TO How_Many
     STEP +2 DO
        GENERIC_LL_STITCH w;
           IF w+2 > How_Many THEN
           BACK_AWAY 450;
               !MoveL Offs(LL_CHAN_WELDS{w,1},0,0,250),V500,Z100,tWeldGun\WObj:=WobJ_FacePlates;
           ENDIF
    ENDFOR
  ENDIF
  THATS_THE_LL_WELDS:
    ENDPROC



    PROC WELD_RL_CHANNEL()


    ActUnit STN1;
    AccSet 100, STOP_DA_SLOP;
    PDispOff;

    MoveJ OFFS(RL_ChanLam_Zs,0,0,250),v1000,Z100,tWeldGun\WObj:=WobJ_FacePlates;

    Search_1D SR_ChanLam_FOUND\SearchStop:=Found_Z, RL_ChanLam_Zs, RL_ChanLam_Ze, V200, tWeldGun\WObj:=WobJ_FacePlates\SchSpeed:=15;
    XnY_Depth RL_ChanLam_Xs, RL_ChanLam_Xe, Found_Z, 23;

    MoveL Offs(RL_ChanLam_Zs,0,0,100),v1000,Z100,tWeldGun\WObj:=WobJ_FacePlates;
    MoveL Offs(RL_Chan_Zs,0,0,100),v1000,Z100,tWeldGun\WObj:=WobJ_FacePlates;

    Search_1D SR_Chan_FOUND\SearchStop:=Found_Z, RL_Chan_Zs, RL_Chan_Ze, V200, tWeldGun\WObj:=WobJ_FacePlates\SchSpeed:=15;
    XnY_Depth RL_Chan_Xs, RL_Chan_Xe, Found_Z, 23;
    SET_CHAN_Zs "RL";

    MoveJ OFFS(RL_Chan_Zs,0,0,250),v1000,Z100,tWeldGun\WObj:=WobJ_FacePlates;
    MoveJ OFFS(RL_ChanLam_Xs,0,0,350),v1000,Z100,tWeldGun\WObj:=WobJ_FacePlates;

    MoveL RelTooL(RL_ChanLam_Xs,0,0,-75),v1000,Z100,tWeldGun\WObj:=WobJ_FacePlates;
    Search_1D SR_ChanLam_FOUND\SearchStop:=Found_ChanLam_X, RL_ChanLam_Xs, RL_ChanLam_Xe, V200, tWeldGun\WObj:=WobJ_FacePlates\SchSpeed:=15;

    MoveL RelTooL(RL_ChanLam_Xs,0,0,-100),v1000,Z100,tWeldGun\WObj:=WobJ_FacePlates;

    MoveL RelTooL(RL_Chan_Xs,0,0,-100),v1000,Z100,tWeldGun\WObj:=WobJ_FacePlates;
    Search_1D SR_Chan_FOUND\SearchStop:=Found_Chan_X, RL_Chan_Xs, RL_Chan_Xe, V200, tWeldGun\WObj:=WobJ_FacePlates\SchSpeed:=15;

    MoveL RelTooL(RL_Chan_Xs,0,0,-250),v1000,Z100,tWeldGun\WObj:=WobJ_FacePlates;
    PDispOff;

    SET_RL_ChanX;

    MoveL Offs(RL_CHAN_WELDS{1,1},0,0,250),v1000,Z100,tWeldGun\WObj:=WobJ_FacePlates;

  IF WeldODDs_Inside_LRnRL = TRUE THEN
    FOR w FROM 1 TO How_Many
     STEP +2 DO
        GENERIC_RL_STITCH w;
           IF w+2 > How_Many THEN
           BACK_AWAY 450;
               !MoveL Offs(RL_CHAN_WELDS{w,1},0,0,250),V500,Z10,tWeldGun\WObj:=WobJ_FacePlates;
           ENDIF
    ENDFOR

  ELSEIF WeldODDs_Inside_LRnRL = FALSE THEN
    FOR w FROM 2 TO How_Many
     STEP +2 DO
        GENERIC_RL_STITCH w;
           IF w+2 > How_Many THEN
           BACK_AWAY 450;
               !MoveL Offs(RL_CHAN_WELDS{w,1},0,0,250),V500,Z10,tWeldGun\WObj:=WobJ_FacePlates;
           ENDIF
    ENDFOR
  ENDIF
!! RIGHT SIDE CHANNEL
MoveJ [[265.54,450.03,360.04],[0.252165,0.224699,-0.93938,-0.0590574],[-1,0,-2,0],[9E+09,-30,180,9E+09,9E+09,9E+09]], v1000, Z50, tWeldGun\WObj:=WobJ_FacePlates;
    THATS_THE_RL_WELDS:
    ENDPROC




PROC WELD_RR_CHANNEL()

    ActUnit STN1;
    AccSet 100, STOP_DA_SLOP;
    PDispOff;

    MoveJ OFFS(RR_ChanLam_Zs,0,0,250),v1000,Z100,tWeldGun\WObj:=WobJ_FacePlates;

    Search_1D SR_ChanLam_FOUND\SearchStop:=Found_Z, RR_ChanLam_Zs, RR_ChanLam_Ze, V200, tWeldGun\WObj:=WobJ_FacePlates\SchSpeed:=15;
    XnY_Depth RR_ChanLam_Xs, RR_ChanLam_Xe, Found_Z, 23;

    MoveL Offs(RR_ChanLam_Zs,0,0,100),v1000,Z100,tWeldGun\WObj:=WobJ_FacePlates;
    MoveL offs(RR_Chan_Zs,0,0,100),v1000,Z100,tWeldGun\WObj:=WobJ_FacePlates;

    Search_1D SR_Chan_FOUND\SearchStop:=Found_Z, RR_Chan_Zs, RR_Chan_Ze, V200, tWeldGun\WObj:=WobJ_FacePlates\SchSpeed:=15;
    XnY_Depth RR_Chan_Xs, RR_Chan_Xe, Found_Z, 23;
    SET_CHAN_Zs "RR";

    MoveL OFFS(RR_Chan_Zs,0,0,250),v1000,Z100,tWeldGun\WObj:=WobJ_FacePlates;
    MoveJ OFFS(RR_ChanLam_Xs,0,0,250),v1000,Z100,tWeldGun\WObj:=WobJ_FacePlates;
    MoveL RelTooL(RR_ChanLam_Xs,0,0,-175),v1000,Z100,tWeldGun\WObj:=WobJ_FacePlates;

    Search_1D SR_ChanLam_FOUND\SearchStop:=Found_ChanLam_X, RR_ChanLam_Xs, RR_ChanLam_Xe, V200, tWeldGun\WObj:=WobJ_FacePlates\SchSpeed:=15;

    MoveL RelTooL(RR_ChanLam_Xs,0,0,-100),v1000,Z100,tWeldGun\WObj:=WobJ_FacePlates;
    MoveL RelTooL(RR_Chan_Xs,0,0,-100),v1000,Z100,tWeldGun\WObj:=WobJ_FacePlates;

    Search_1D SR_Chan_FOUND\SearchStop:=Found_Chan_X, RR_Chan_Xs, RR_Chan_Xe, V200, tWeldGun\WObj:=WobJ_FacePlates\SchSpeed:=15;

    MoveL RelTooL(RR_Chan_Xs,0,0,-150),v1000,Z100,tWeldGun\WObj:=WobJ_FacePlates;
    PDispOff;
    SET_RR_ChanX;

    MoveL Offs(RR_CHAN_WELDS{1,1},0,0,250),v1000,Z100,tWeldGun\WObj:=WobJ_FacePlates;

  IF WeldEVENs_Outside_LLnRR = TRUE THEN
    FOR w FROM 2 TO How_Many
     STEP +2 DO
        GENERIC_RR_STITCH w;
           IF w+2 > How_Many THEN
           BACK_AWAY 450;
               !MoveL Offs(RR_CHAN_WELDS{w,1},0,0,250),V500,Z100,tWeldGun\WObj:=WobJ_FacePlates;
           ENDIF
    ENDFOR

  ELSEIF WeldEVENs_Outside_LLnRR = FALSE THEN
    FOR w FROM 1 TO How_Many
     STEP +2 DO
        GENERIC_RR_STITCH w;
           IF w+2 > How_Many THEN
           BACK_AWAY 450;
               !MoveL Offs(RR_CHAN_WELDS{w,1},0,0,250),V500,Z100,tWeldGun\WObj:=WobJ_FacePlates;
           ENDIF
    ENDFOR
  ENDIF
THATS_THE_RR_WELDS:
ENDPROC



PROC WELD_LR_CHANNEL()

    ActUnit STN1;
    AccSet 100, STOP_DA_SLOP;
    PDispOff;

    MoveJ OFFS(LR_ChanLam_Zs,0,0,250),v1000,Z100,tWeldGun\WObj:=WobJ_FacePlates;

    Search_1D SR_ChanLam_FOUND\SearchStop:=Found_Z, LR_ChanLam_Zs, LR_ChanLam_Ze, v200, tWeldGun\WObj:=WobJ_FacePlates\SchSpeed:=15;
    XnY_Depth LR_ChanLam_Xs, LR_ChanLam_Xe, Found_Z, 23;

    MoveL offs(LR_ChanLam_Zs,0,0,100),v1000,Z100,tWeldGun\WObj:=WobJ_FacePlates;
    MoveL offs(LR_Chan_Zs,0,0,100),v1000,Z100,tWeldGun\WObj:=WobJ_FacePlates;

    Search_1D SR_Chan_FOUND\SearchStop:=Found_Z, LR_Chan_Zs, LR_Chan_Ze, v200, tWeldGun\WObj:=WobJ_FacePlates\SchSpeed:=15;
    XnY_Depth LR_Chan_Xs, LR_Chan_Xe, Found_Z, 23;
    SET_CHAN_Zs "LR";

    MoveL offs(LR_Chan_Zs,0,0,100),v1000,Z100,tWeldGun\WObj:=WobJ_FacePlates;
    MoveJ OFFS(LR_ChanLam_Xs,0,0,350),v1000,Z100,tWeldGun\WObj:=WobJ_FacePlates;
    MoveL RelTooL(LR_ChanLam_Xs,0,0,-75),v1000,Z100,tWeldGun\WObj:=WobJ_FacePlates;

    Search_1D SR_ChanLam_FOUND\SearchStop:=Found_ChanLam_X, LR_ChanLam_Xs, LR_ChanLam_Xe, v200, tWeldGun\WObj:=WobJ_FacePlates\SchSpeed:=15;

    MoveL RelTooL(LR_ChanLam_Xs,0,0,-100),v1000,Z100,tWeldGun\WObj:=WobJ_FacePlates;
    MoveL RelTooL(LR_Chan_Xs,0,0,-100),v1000,Z100,tWeldGun\WObj:=WobJ_FacePlates;

    Search_1D SR_Chan_FOUND\SearchStop:=Found_Chan_X, LR_Chan_Xs, LR_Chan_Xe, v200, tWeldGun\WObj:=WobJ_FacePlates\SchSpeed:=15;

    MoveL RelTooL(LR_Chan_Xs,0,0,-250),v1000,Z100,tWeldGun\WObj:=WobJ_FacePlates;

    PDispOff;
    SET_LR_ChanX;
    MoveL Offs(LR_CHAN_WELDS{1,1},0,0,250),v1000,Z100,tWeldGun\WObj:=WobJ_FacePlates;

  IF WeldODDs_Inside_LRnRL = TRUE THEN
    FOR w FROM 1 TO How_Many
     STEP +2 DO
        GENERIC_LR_STITCH w;
           IF w+2 > How_Many THEN
            BACK_AWAY 450;
               !MoveL Offs(LR_CHAN_WELDS{w,1},0,0,250),V500,Z100,tWeldGun\WObj:=WobJ_FacePlates;
           ENDIF
    ENDFOR

  ELSEIF WeldODDs_Inside_LRnRL = FALSE THEN
    FOR w FROM 2 TO How_Many
     STEP +2 DO
        GENERIC_LR_STITCH w;
           IF w+2 > How_Many THEN
           BACK_AWAY 450;
               ! MoveL Offs(LR_CHAN_WELDS{w,1},0,0,250),V500,Z100,tWeldGun\WObj:=WobJ_FacePlates;
           ENDIF
    ENDFOR
  ENDIF
    THATS_THE_LR_WELDS:
    PDispOff;
ENDPROC




PROC SET_LL_ChanX()

 FOR i FROM 1 TO HOW_MANY
    STEP +1 DO
       FOR j FROM 1 TO 3
       STEP +1 DO

    SET_X_CHAN_LnR "LL", LL_CHAN_WELDS{i,j}, Found_Chan_X,Found_ChanLam_X;
    ENDFOR
 ENDFOR
    waittime\inpos,.01;
ENDPROC


PROC SET_LR_ChanX()

FOR i FROM 1 TO HOW_MANY
  STEP +1 DO
    FOR j FROM 1 TO 3
      STEP +1 DO

    SET_X_CHAN_LnR "LR", LR_CHAN_WELDS{i,j}, Found_Chan_X,Found_ChanLam_X;
    ENDFOR
ENDFOR
    waittime\inpos,.01;
ENDPROC


PROC SET_RL_ChanX()

FOR i FROM 1 TO HOW_MANY
  STEP +1 DO
    FOR j FROM 1 TO 3
      STEP +1 DO

    SET_X_CHAN_LnR "RL", RL_CHAN_WELDS{i,j}, Found_Chan_X,Found_ChanLam_X;
    waittime\inpos,.01;

    ENDFOR
ENDFOR
ENDPROC


PROC SET_RR_ChanX()
FOR i FROM 1 TO HOW_MANY
  STEP +1 DO
    FOR j FROM 1 TO 3
      STEP +1 DO

    SET_X_CHAN_LnR "RR", RR_CHAN_WELDS{i,j}, Found_Chan_X,Found_ChanLam_X;
    ENDFOR
ENDFOR
    waittime\inpos,.01;
ENDPROC



    PROC SET_X_CHAN_LnR(
    STRING WHAT_SIDE,
    INOUT ROBTARGET The_Weld,
    INOUT ROBTARGET Chan_Found,
    INOUT ROBTARGET ChanLam_FOUND)
!!notes 1/14/19 added Top_Of_Chan_Y for when its less than 3 cross bars
!    VAR num Top_Of_Chan_Y :=0;

!        IF HORIZ_Y3 > 0 and HORIZ_Y3 = FP_Height THEN
!            Top_Of_Chan_Y := HORIZ_Y3;
!        ELSEIF HORIZ_Y3 = 0 AND HORIZ_Y2 = FP_Height THEN
!            Top_Of_Chan_Y := HORIZ_Y2;
!        ELSEIF HORIZ_Y3 = 0 AND HORIZ_Y2 = 0 and HORIZ_Y1 = FP_Height THEN
!            Top_Of_Chan_Y := HORIZ_Y1;
!        ELSEIF HORIZ_Y3 > 0 AND HORIZ_Y2 > 0 and HORIZ_Y1 > 0 AND HORIZ_Y4 = FP_Height THEN
!            Top_Of_Chan_Y := HORIZ_Y4;
!            ENDIF
    IF WHAT_SIDE = "LL" THEN

        IF The_Weld.trans.Y < Lam_OverLap THEN
               The_Weld.trans.X := ChanLam_FOUND.trans.X + Minor_Nozzle_Radius - (FP_StickOut * 1.15);

        ELSEIF The_Weld.trans.Y >= Lam_OverLap THEN
               The_Weld.trans.X := Chan_FOUND.trans.X + Minor_Nozzle_Radius - (FP_StickOut * 1.15 );
        ENDIF

    ELSEIF WHAT_SIDE = "LR" THEN

            IF The_Weld.trans.Y < (Top_Of_Chan_Y - CHANNEL_LENGTH)  THEN
                The_Weld.trans.X := ChanLam_FOUND.trans.X + Minor_Nozzle_Radius + BAR_THICKNESS + FP_StickOut ;

            ELSEIF The_Weld.trans.Y >= (Top_Of_Chan_Y - CHANNEL_LENGTH) AND The_Weld.trans.Y <= Top_Of_Chan_Y  THEN
                The_Weld.trans.X := Chan_FOUND.trans.X + Minor_Nozzle_Radius + CHANNEL_WIDTH + FP_StickOut ;

            ELSEIF The_Weld.trans.Y > Top_Of_Chan_Y THEN
                The_Weld.trans.X := Chan_FOUND.trans.X + Minor_Nozzle_Radius + BAR_THICKNESS + FP_StickOut ;

            ENDIF

    ELSEIF WHAT_SIDE = "RR" THEN

        IF The_Weld.trans.Y < Lam_OverLap THEN
               The_Weld.trans.X := ChanLam_FOUND.trans.X - Minor_Nozzle_Radius + (FP_StickOut * 1.15) ;

        ELSEIF The_Weld.trans.Y > Lam_OverLap   THEN
               The_Weld.trans.X := Chan_FOUND.trans.X - Minor_Nozzle_Radius + (FP_StickOut * 1.15) ;

        ENDIF

    ELSEIF WHAT_SIDE = "RL" THEN

            IF The_Weld.trans.Y < (Top_Of_Chan_Y - CHANNEL_LENGTH) THEN
                The_Weld.trans.X := ChanLam_FOUND.trans.X - Minor_Nozzle_Radius - BAR_THICKNESS - FP_StickOut;

            ELSEIF The_Weld.trans.Y >= (Top_Of_Chan_Y - CHANNEL_LENGTH) AND The_Weld.trans.Y < Top_Of_Chan_Y THEN
                The_Weld.trans.X := Chan_FOUND.trans.X - Minor_Nozzle_Radius - CHANNEL_WIDTH - FP_StickOut;

           ELSEIF The_Weld.trans.Y > Top_Of_Chan_Y THEN
                The_Weld.trans.X := Chan_FOUND.trans.X - Minor_Nozzle_Radius - BAR_THICKNESS - FP_StickOut;
            ENDIF

    ENDIF
        WAITTIME\INPOS,.1;
            ENDPROC







   PROC SET_CHAN_Zs(
    STRING PICK_UH_CHAN)

    IF PICK_UH_CHAN = "RL" THEN
       FOR i FROM 1 TO HOW_MANY
       STEP +1 DO
        CHAN_Z_SET_DEPTH RL_CHAN_WELDS{i,1}, RL_CHAN_WELDS{i,2}, RL_CHAN_WELDS{i,3}, CHAN_Found_Z, CHANLAM_Found_Z ;
       ENDFOR

    ELSEIF PICK_UH_CHAN = "LR" THEN
       FOR f FROM 1 TO HOW_MANY
       STEP +1 DO
        CHAN_Z_SET_DEPTH LR_CHAN_WELDS{f,1}, LR_CHAN_WELDS{f,2}, LR_CHAN_WELDS{f,3}, CHAN_Found_Z, CHANLAM_Found_Z ;
       ENDFOR

    ELSEIF PICK_UH_CHAN = "RR" THEN
       FOR g FROM 1 TO HOW_MANY
       STEP +1 DO
        CHAN_Z_SET_DEPTH RR_CHAN_WELDS{g,1}, RR_CHAN_WELDS{g,2}, RR_CHAN_WELDS{g,3}, CHAN_Found_Z, CHANLAM_Found_Z ;
       ENDFOR

    ELSEIF PICK_UH_CHAN = "LL" THEN
       FOR a FROM 1 TO HOW_MANY
       STEP +1 DO
        CHAN_Z_SET_DEPTH LL_CHAN_WELDS{a,1}, LL_CHAN_WELDS{a,2}, LL_CHAN_WELDS{a,3}, CHAN_Found_Z, CHANLAM_Found_Z ;
       ENDFOR

    ENDIF
    THAT_SET_IT:
    ENDPROC





    PROC GENERIC_RL_STITCH(
         NUM RL_WELD)

IF RL_CHAN_NOTES{RL_WELD,1} = "SKIP" OR ( RL_WELD = 1 and Anchor_Y <= 75) THEN GOTO No_Weld_Here; ENDIF
    MoveL Offs(RL_CHAN_WELDS{RL_WELD,1},0,0,125),V500,Z50,tWeldGun\WObj:=WobJ_FacePlates;
    MoveL RelTooL(RL_CHAN_WELDS{RL_WELD,1},0,0,-50),V500,Z10,tWeldGun\WObj:=WobJ_FacePlates;
    TPWrite RL_CHAN_NOTES{RL_WELD,1};
    TPWrite RL_CHAN_NOTES{RL_WELD,2};

    WArcLStart RL_CHAN_WELDS{RL_WELD,1},v100,SE_CHANNEL,BD_CHANNEL,Z1,tWeldGun\WObj:=WobJ_FacePlates\Track:=TRK_CHANNEL;
IF RL_CHAN_NOTES {RL_WELD,1}= "CORNER" THEN
    WArcL RL_CHAN_WELDS{RL_WELD,2}, v100, z10, tWeldGun\WObj:=WobJ_FacePlates\Track:=TRK_CHANNEL;
ENDIF
    WArcLEnd RL_CHAN_WELDS{RL_WELD,3}, v100, z1, tWeldGun\WObj:=WobJ_FacePlates\Track:=TRK_CHANNEL;

    MoveL RelTooL(RL_CHAN_WELDS{RL_WELD,3},0,0,-50),V500,Z10,tWeldGun\WObj:=WobJ_FacePlates;
    MoveL Offs(RL_CHAN_WELDS{RL_WELD,3},0,0,125),V500,Z50,tWeldGun\WObj:=WobJ_FacePlates;
    No_Weld_Here:
    ENDPROC





    PROC GENERIC_LL_STITCH(
          NUM LL_WELD)
!IF Y1_TightBox = TRUE AND WeldEVENs_Outside_LLnRR = FALSE AND LL_WELD = 1 THEN GOTO No_Weld_Here; ENDIF
IF LL_CHAN_NOTES{LL_WELD,1} = "SKIP" THEN GOTO No_Weld_Here; ENDIF

    MoveL Offs(LL_CHAN_WELDS{LL_WELD,1},0,0,125),V500,Z50,tWeldGun\WObj:=WobJ_FacePlates;
    MoveL RelTooL(LL_CHAN_WELDS{LL_WELD,1},0,0,-50),V500,Z10,tWeldGun\WObj:=WobJ_FacePlates;

    WArcLStart LL_CHAN_WELDS{LL_WELD,1},v100,SE_CHANNEL,BD_CHANNEL,Z1,tWeldGun\WObj:=WobJ_FacePlates\Track:=TRK_CHANNEL;
IF LL_CHAN_NOTES {LL_WELD,1}= "CORNER" THEN
    WArcL LL_CHAN_WELDS{LL_WELD,2}, v100, z10, tWeldGun\WObj:=WobJ_FacePlates\Track:=TRK_CHANNEL;
ENDIF
    WArcLEnd LL_CHAN_WELDS{LL_WELD,3}, v100, z1, tWeldGun\WObj:=WobJ_FacePlates\Track:=TRK_CHANNEL;

    MoveL RelTooL(LL_CHAN_WELDS{LL_WELD,3},0,0,-50),V500,Z10,tWeldGun\WObj:=WobJ_FacePlates;
    MoveL RelTooL(LL_CHAN_WELDS{LL_WELD,3},0,0,-75),V500,Z50,tWeldGun\WObj:=WobJ_FacePlates;
    MoveL Offs(LL_CHAN_WELDS{LL_WELD,3},0,0,125),V500,Z50,tWeldGun\WObj:=WobJ_FacePlates;

    No_Weld_Here:
    ENDPROC





    PROC GENERIC_LR_STITCH(
         NUM LR_WELD)

IF LR_CHAN_NOTES{LR_WELD,1} = "SKIP" OR ( LR_WELD = 1 and Anchor_Y <= 75) THEN GOTO No_Weld_Here; ENDIF

    MoveL Offs(LR_CHAN_WELDS{LR_WELD,1},0,0,125),V500,Z50,tWeldGun\WObj:=WobJ_FacePlates;
    MoveL RelTooL(LR_CHAN_WELDS{LR_WELD,1},0,0,-75),V500,Z20,tWeldGun\WObj:=WobJ_FacePlates;
    MoveL RelTooL(LR_CHAN_WELDS{LR_WELD,1},0,0,-50),V500,Z10,tWeldGun\WObj:=WobJ_FacePlates;

    WArcLStart LR_CHAN_WELDS{LR_WELD,1},v100,SE_CHANNEL,BD_CHANNEL,Z1,tWeldGun\WObj:=WobJ_FacePlates\Track:=TRK_CHANNEL;
IF LR_CHAN_NOTES {LR_WELD,1}= "CORNER" THEN
        WArcL LR_CHAN_WELDS{LR_WELD,2}, v100, z10, tWeldGun\WObj:=WobJ_FacePlates\Track:=TRK_CHANNEL;
ENDIF
    WArcLEnd LR_CHAN_WELDS{LR_WELD,3}, v100, z1, tWeldGun\WObj:=WobJ_FacePlates\Track:=TRK_CHANNEL;

    MoveL RelTooL(LR_CHAN_WELDS{LR_WELD,3},0,0,-75),V500,Z10,tWeldGun\WObj:=WobJ_FacePlates;
    MoveL Offs(LR_CHAN_WELDS{LR_WELD,3},0,0,125),V500,Z50,tWeldGun\WObj:=WobJ_FacePlates;

    No_Weld_Here:
    ENDPROC





    PROC GENERIC_RR_STITCH(
         NUM RR_WELD)
!IF Y1_TightBox = TRUE AND WeldEVENs_Outside_LLnRR = FALSE AND RR_WELD = 1 THEN GOTO No_Weld_Here; ENDIF
IF  RR_CHAN_NOTES{RR_WELD,1} = "SKIP" THEN GOTO No_Weld_Here; ENDIF

    MoveL Offs(RR_CHAN_WELDS{RR_WELD,1},0,0,150),V500,Z50,tWeldGun\WObj:=WobJ_FacePlates;
    MoveL RelTooL(RR_CHAN_WELDS{RR_WELD,1},0,0,-75),V500,Z20,tWeldGun\WObj:=WobJ_FacePlates;
    MoveL RelTooL(RR_CHAN_WELDS{RR_WELD,1},0,0,-50),V500,Z10,tWeldGun\WObj:=WobJ_FacePlates;

    WArcLStart RR_CHAN_WELDS{RR_WELD,1},v100,SE_CHANNEL,BD_CHANNEL,Z1,tWeldGun\WObj:=WobJ_FacePlates\Track:=TRK_CHANNEL;
IF RR_CHAN_NOTES {RR_WELD,1}= "CORNER" THEN
    WArcL RR_CHAN_WELDS{RR_WELD,2}, v100, z10, tWeldGun\WObj:=WobJ_FacePlates\Track:=TRK_CHANNEL;
ENDIF
    WArcLEnd RR_CHAN_WELDS{RR_WELD,3}, v100, z1, tWeldGun\WObj:=WobJ_FacePlates\Track:=TRK_CHANNEL;

    MoveL RelTooL(RR_CHAN_WELDS{RR_WELD,3},0,0,-75),V500,Z10,tWeldGun\WObj:=WobJ_FacePlates;
    MoveL Offs(RR_CHAN_WELDS{RR_WELD,3},0,0,150),V500,Z50,tWeldGun\WObj:=WobJ_FacePlates;

No_Weld_Here:
ENDPROC




PROC ALL_Chan_Plan(NUM WELD_LENGTH)


IF LOAD_PUSH = TRUE  THEN
    OAL_Stitch :=  FP_Height - FP_Thickness - (2*FP_StickOut);
ELSEIF LOAD_PUSH = FALSE THEN
    OAL_Stitch := FP_Height - ( HORIZ_Y2 + bar_thickness + (2*FP_StickOut));
ENDIF

How_Many := ROUND( OAL_Stitch / WELD_LENGTH );
How_Long := OAL_Stitch / How_Many;
FROM_HERE := FP_Height - OAL_Stitch - fp_stickout;
TPErase;
TPWrite" How_Many :="\Num:=How_Many;
TPWrite" How_Long := "\Num:=How_Long;

    FOR k FROM 1 TO How_Many
    STEP + 1 DO

    IF K = 1 THEN
     LL_CHAN_WELDS{ k , 1}.trans.Y :=  FROM_HERE + ( k * How_Long ) ;
     LL_CHAN_WELDS{ k , 1}.EXTAX := LL_CHAN_GOINGdown.extax;
     LL_CHAN_WELDS{ k , 1}.ROT := LL_CHAN_GOINGdown.ROT;
     LL_CHAN_WELDS{ k , 1}.RobConf := LL_CHAN_GOINGdown.RobConf;

     IF LOAD_PUSH = FALSE THEN
     LL_CHAN_WELDS{ k , 2}.trans.Y :=  FROM_HERE + ( k * How_Long ) - How_Long + NOZZLE_RADIUS ;
     LL_CHAN_WELDS{ k , 2}.EXTAX := LL_CHAN_GOINGdown.extax;
     LL_CHAN_WELDS{ k , 2}.ROT := LL_CHAN_GOINGdown.ROT;
     LL_CHAN_WELDS{ k , 2}.RobConf := LL_CHAN_GOINGdown.RobConf;
     ELSEIF LOAD_PUSH = TRUE THEN
     LL_CHAN_WELDS{ k , 2}.trans.Y :=  FROM_HERE + ( k * How_Long ) - How_Long + NOZZLE_RADIUS ;
     LL_CHAN_WELDS{ k , 2}.EXTAX := LL_CHAN_GOINGdown.extax;
     LL_CHAN_WELDS{ k , 2}.ROT := LL_CHAN_GOINGdownCORNER.ROT;
     LL_CHAN_WELDS{ k , 2}.RobConf := LL_CHAN_GOINGdownCORNER.RobConf;
     ENDIF

     LL_CHAN_WELDS{ k , 3}.trans.Y :=  FROM_HERE + ( k * How_Long ) - How_Long ;
     LL_CHAN_WELDS{ k , 3}.EXTAX := LL_CHAN_GOINGdownCORNER.extax;
     LL_CHAN_WELDS{ k , 3}.ROT := LL_CHAN_GOINGdownCORNER.ROT;
     LL_CHAN_WELDS{ k , 3}.RobConf := LL_CHAN_GOINGdownCORNER.RobConf;
!!$$$$$$$$$
     LR_CHAN_WELDS{ k , 1}.trans.Y :=  FROM_HERE + ( k * How_Long ) ;
     LR_CHAN_WELDS{ k , 1}.EXTAX := LR_CHAN_GOINGdown.extax;
     LR_CHAN_WELDS{ k , 1}.ROT := LR_CHAN_GOINGdown.ROT;
     LR_CHAN_WELDS{ k , 1}.RobConf := LR_CHAN_GOINGdown.RobConf;

     IF LOAD_PUSH = FALSE THEN
     LR_CHAN_WELDS{ k , 2}.trans.Y :=  FROM_HERE + ( k * How_Long ) - How_Long + NOZZLE_RADIUS ;
     LR_CHAN_WELDS{ k , 2}.EXTAX := LR_CHAN_GOINGdown.extax;
     LR_CHAN_WELDS{ k , 2}.ROT := LR_CHAN_GOINGdown.ROT;
     LR_CHAN_WELDS{ k , 2}.RobConf := LR_CHAN_GOINGdown.RobConf;
     ELSEIF LOAD_PUSH = TRUE THEN
     LR_CHAN_WELDS{ k , 2}.trans.Y :=  FROM_HERE + ( k * How_Long ) - How_Long + NOZZLE_RADIUS ;
     LR_CHAN_WELDS{ k , 2}.EXTAX := LR_CHAN_GOINGdown.extax;
     LR_CHAN_WELDS{ k , 2}.ROT := LR_CHAN_GOINGdown_CORNER.ROT;
     LR_CHAN_WELDS{ k , 2}.RobConf := LR_CHAN_GOINGdown_CORNER.RobConf;
     ENDIF

     LR_CHAN_WELDS{ k , 3}.trans.Y :=  FROM_HERE + ( k * How_Long ) - How_Long ;
     LR_CHAN_WELDS{ k , 3}.EXTAX := LR_CHAN_GOINGdown_CORNER.extax;
     LR_CHAN_WELDS{ k , 3}.ROT := LR_CHAN_GOINGdown_CORNER.ROT;
     LR_CHAN_WELDS{ k , 3}.RobConf := LR_CHAN_GOINGdown_CORNER.RobConf;

!!$$$$$$$$$
     RR_CHAN_WELDS{ k , 1}.trans.Y :=  FROM_HERE + ( k * How_Long ) ;
     RR_CHAN_WELDS{ k , 1}.EXTAX := RR_CHAN_GOINGdown.extax;
     RR_CHAN_WELDS{ k , 1}.ROT := RR_CHAN_GOINGdown.ROT;
     RR_CHAN_WELDS{ k , 1}.RobConf := RR_CHAN_GOINGdown.RobConf;

     IF LOAD_PUSH = FALSE THEN
     RR_CHAN_WELDS{ k , 2}.trans.Y :=  FROM_HERE + ( k * How_Long ) - How_Long + NOZZLE_RADIUS ;
     RR_CHAN_WELDS{ k , 2}.EXTAX := RR_CHAN_GOINGdown.extax;
     RR_CHAN_WELDS{ k , 2}.ROT := RR_CHAN_GOINGdown.ROT;
     RR_CHAN_WELDS{ k , 2}.RobConf := RR_CHAN_GOINGdown.RobConf;
     ELSEIF LOAD_PUSH = TRUE THEN
     RR_CHAN_WELDS{ k , 2}.trans.Y :=  FROM_HERE + ( k * How_Long ) - How_Long + NOZZLE_RADIUS ;
     RR_CHAN_WELDS{ k , 2}.EXTAX := RR_CHAN_GOINGdown.extax;
     RR_CHAN_WELDS{ k , 2}.ROT := RR_CHAN_BOTTOMcorner.ROT;
     RR_CHAN_WELDS{ k , 2}.RobConf := RR_CHAN_BOTTOMcorner.RobConf;
     ENDIF

     RR_CHAN_WELDS{ k , 3}.trans.Y :=  FROM_HERE + ( k * How_Long ) - How_Long ;
     RR_CHAN_WELDS{ k , 3}.EXTAX := RR_CHAN_BOTTOMcorner.extax;
     RR_CHAN_WELDS{ k , 3}.ROT := RR_CHAN_BOTTOMcorner.ROT;
     RR_CHAN_WELDS{ k , 3}.RobConf := RR_CHAN_BOTTOMcorner.RobConf;
!!$$$$$$$$$
     RL_CHAN_WELDS{ k , 1}.trans.Y :=  FROM_HERE + ( k * How_Long ) ;
     RL_CHAN_WELDS{ k , 1}.EXTAX := RL_CHAN_GOINGdown.extax;
     RL_CHAN_WELDS{ k , 1}.ROT := RL_CHAN_GOINGdown.ROT;
     RL_CHAN_WELDS{ k , 1}.RobConf := RL_CHAN_GOINGdown.RobConf;

     IF LOAD_PUSH = FALSE THEN
     RL_CHAN_WELDS{ k , 2}.trans.Y :=  FROM_HERE + ( k * How_Long ) - How_Long + NOZZLE_RADIUS ;
     RL_CHAN_WELDS{ k , 2}.EXTAX := RL_CHAN_GOINGdown.extax;
     RL_CHAN_WELDS{ k , 2}.ROT := RL_CHAN_GOINGdown.ROT;
     RL_CHAN_WELDS{ k , 2}.RobConf := RL_CHAN_GOINGdown.RobConf;
     ELSEIF LOAD_PUSH = TRUE THEN
     RL_CHAN_WELDS{ k , 2}.trans.Y :=  FROM_HERE + ( k * How_Long ) - How_Long + NOZZLE_RADIUS ;
     RL_CHAN_WELDS{ k , 2}.EXTAX := RL_CHAN_GOINGdown.extax;
     RL_CHAN_WELDS{ k , 2}.ROT := RL_Chan_BOTTOMcorner.ROT;
     RL_CHAN_WELDS{ k , 2}.RobConf := RL_Chan_BOTTOMcorner.RobConf;
     ENDIF

     RL_CHAN_WELDS{ k , 3}.trans.Y :=  FROM_HERE + ( k * How_Long ) - How_Long ;
     RL_CHAN_WELDS{ k , 3}.EXTAX := RL_Chan_BOTTOMcorner.extax;
     RL_CHAN_WELDS{ k , 3}.ROT := RL_Chan_BOTTOMcorner.ROT;
     RL_CHAN_WELDS{ k , 3}.RobConf := RL_Chan_BOTTOMcorner.RobConf;
!!$$$$$$$$$
     RR_CHAN_NOTES{ k , 1}:="CORNER";
     RL_CHAN_NOTES{ k , 1}:="CORNER";
     LR_CHAN_NOTES{ k , 1}:="CORNER";
     LL_CHAN_NOTES{ k , 1}:="CORNER";
!!$$$$$$$$$

    ELSEIF k <> 1 AND k < How_Many THEN
     LL_CHAN_WELDS{ k , 1}.trans.Y :=  FROM_HERE + ( k * How_Long ) - How_Long;
     LL_CHAN_WELDS{ k , 1}.EXTAX := LL_CHAN_GoingUp.extax;
     LL_CHAN_WELDS{ k , 1}.ROT := LL_CHAN_GoingUp.ROT;
     LL_CHAN_WELDS{ k , 1}.RobConf := LL_CHAN_GoingUp.RobConf;

     LL_CHAN_WELDS{ k , 2}.trans.Y :=  FROM_HERE + ( k * How_Long ) - NOZZLE_RADIUS ;
     LL_CHAN_WELDS{ k , 2}.EXTAX := LL_CHAN_GoingUp.extax;
     LL_CHAN_WELDS{ k , 2}.ROT := LL_CHAN_GoingUp.ROT;
     LL_CHAN_WELDS{ k , 2}.RobConf := LL_CHAN_GoingUp.RobConf;

     LL_CHAN_WELDS{ k , 3}.trans.Y :=  FROM_HERE + ( k * How_Long );
     LL_CHAN_WELDS{ k , 3}.EXTAX := LL_CHAN_GoingUp.extax;
     LL_CHAN_WELDS{ k , 3}.ROT := LL_CHAN_GoingUp.ROT;
     LL_CHAN_WELDS{ k , 3}.RobConf := LL_CHAN_GoingUp.RobConf;

!!$$$$$$$$$

     LR_CHAN_WELDS{ k , 1}.trans.Y :=  FROM_HERE + ( k * How_Long ) - How_Long;
     IF LR_CHAN_WELDS{ k , 1}.trans.Y < (Top_Of_Chan_Y - CHANNEL_LENGTH) OR LR_CHAN_WELDS{ k , 1}.trans.Y > Top_Of_Chan_Y THEN
        LR_CHAN_WELDS{ k , 1}.EXTAX := LR_CHAN_GOINGup.extax;
        LR_CHAN_WELDS{ k , 1}.ROT := LR_CHAN_GOINGup.ROT;
        LR_CHAN_WELDS{ k , 1}.RobConf := LR_CHAN_GOINGup.RobConf;
     ELSEIF LR_CHAN_WELDS{ k , 1}.trans.Y > (Top_Of_Chan_Y - CHANNEL_LENGTH) AND LR_CHAN_WELDS{ k , 1}.trans.Y < Top_Of_Chan_Y THEN
        LR_CHAN_WELDS{ k , 1}.EXTAX := LR_CHANFLAT_GOINGup.extax;
        LR_CHAN_WELDS{ k , 1}.ROT := LR_CHANFLAT_GOINGup.ROT;
        LR_CHAN_WELDS{ k , 1}.RobConf := LR_CHANFLAT_GOINGup.RobConf;
     ENDIF

